LIN {X 266.912,Y -113.394,Z 120.558,A 156.982,B 90.000,C 0.000} C_DIS
LIN {X 267.031,Y -113.112,Z 120.601,A 157.043,B 90.000,C 0.000} C_DIS
LIN {X 267.056,Y -113.053,Z 120.652,A 157.056,B 90.000,C 0.000} C_DIS
LIN {X 267.089,Y -112.975,Z 120.703,A 157.072,B 90.000,C 0.000} C_DIS
LIN {X 267.248,Y -112.599,Z 120.745,A 157.153,B 90.000,C 0.000} C_DIS
LIN {X 267.281,Y -112.521,Z 120.796,A 157.170,B 90.000,C 0.000} C_DIS
LIN {X 267.306,Y -112.462,Z 120.847,A 157.182,B 90.000,C 0.000} C_DIS
LIN {X 267.424,Y -112.180,Z 120.890,A 157.243,B 90.000,C 0.000} C_DIS
LIN {X 267.449,Y -112.121,Z 120.941,A 157.255,B 90.000,C 0.000} C_DIS
LIN {X 267.482,Y -112.043,Z 120.992,A 157.272,B 90.000,C 0.000} C_DIS
LIN {X 267.639,Y -111.666,Z 121.034,A 157.353,B 90.000,C 0.000} C_DIS
LIN {X 267.705,Y -111.509,Z 121.137,A 157.386,B 90.000,C 0.000} C_DIS
LIN {X 267.861,Y -111.132,Z 121.179,A 157.467,B 90.000,C 0.000} C_DIS
LIN {X 267.894,Y -111.054,Z 121.230,A 157.484,B 90.000,C 0.000} C_DIS
LIN {X 267.918,Y -110.995,Z 121.281,A 157.496,B 90.000,C 0.000} C_DIS
LIN {X 268.035,Y -110.712,Z 121.324,A 157.557,B 90.000,C 0.000} C_DIS
LIN {X 268.060,Y -110.653,Z 121.375,A 157.570,B 90.000,C 0.000} C_DIS
LIN {X 268.092,Y -110.574,Z 121.426,A 157.586,B 90.000,C 0.000} C_DIS
LIN {X 268.247,Y -110.197,Z 121.468,A 157.667,B 90.000,C 0.000} C_DIS
LIN {X 268.312,Y -110.040,Z 121.570,A 157.701,B 90.000,C 0.000} C_DIS
LIN {X 268.466,Y -109.662,Z 121.613,A 157.781,B 90.000,C 0.000} C_DIS
LIN {X 268.499,Y -109.583,Z 121.664,A 157.798,B 90.000,C 0.000} C_DIS
LIN {X 268.523,Y -109.524,Z 121.715,A 157.811,B 90.000,C 0.000} C_DIS
LIN {X 268.638,Y -109.241,Z 121.757,A 157.871,B 90.000,C 0.000} C_DIS
LIN {X 268.662,Y -109.182,Z 121.808,A 157.884,B 90.000,C 0.000} C_DIS
LIN {X 268.694,Y -109.103,Z 121.859,A 157.900,B 90.000,C 0.000} C_DIS
LIN {X 268.847,Y -108.725,Z 121.902,A 157.981,B 90.000,C 0.000} C_DIS
LIN {X 268.879,Y -108.646,Z 121.953,A 157.998,B 90.000,C 0.000} C_DIS
LIN {X 268.899,Y -108.596,Z 122.004,A 158.009,B 90.000,C 0.000} C_DIS
LIN {X 269.023,Y -108.291,Z 122.077,A 158.074,B 90.000,C 0.000} C_DIS
LIN {X 269.087,Y -108.131,Z 122.214,A 158.108,B 90.000,C 0.000} C_DIS
LIN {X 269.132,Y -108.018,Z 122.410,A 158.132,B 90.000,C 0.000} C_DIS
LIN {X 269.157,Y -107.956,Z 122.817,A 158.145,B 90.000,C 0.000} C_DIS
LIN {X 269.176,Y -107.909,Z 122.892,A 158.155,B 90.000,C 0.000} C_DIS
LIN {X 269.195,Y -107.861,Z 123.037,A 158.165,B 90.000,C 0.000} C_DIS
LIN {X 269.211,Y -107.822,Z 123.759,A 158.173,B 90.000,C 0.000} C_DIS
LIN {X 269.249,Y -107.726,Z 124.048,A 158.194,B 90.000,C 0.000} C_DIS
LIN {X 269.264,Y -107.688,Z 124.771,A 158.202,B 90.000,C 0.000} C_DIS
LIN {X 269.303,Y -107.592,Z 125.060,A 158.222,B 90.000,C 0.000} C_DIS
LIN {X 269.318,Y -107.554,Z 125.783,A 158.230,B 90.000,C 0.000} C_DIS
LIN {X 269.356,Y -107.458,Z 126.072,A 158.251,B 90.000,C 0.000} C_DIS
LIN {X 269.372,Y -107.420,Z 126.794,A 158.259,B 90.000,C 0.000} C_DIS
LIN {X 269.391,Y -107.372,Z 126.939,A 158.269,B 90.000,C 0.000} C_DIS
LIN {X 269.410,Y -107.324,Z 127.003,A 158.279,B 90.000,C 0.000} C_DIS
LIN {X 269.431,Y -107.271,Z 127.336,A 158.291,B 90.000,C 0.000} C_DIS
LIN {X 269.498,Y -107.103,Z 127.372,A 158.326,B 90.000,C 0.000} C_DIS
LIN {X 269.554,Y -106.961,Z 127.351,A 158.356,B 90.000,C 0.000} C_DIS
LIN {X 269.601,Y -106.842,Z 127.249,A 158.382,B 90.000,C 0.000} C_DIS
LIN {X 269.714,Y -106.558,Z 127.207,A 158.442,B 90.000,C 0.000} C_DIS
LIN {X 269.760,Y -106.439,Z 127.105,A 158.467,B 90.000,C 0.000} C_DIS
LIN {X 269.873,Y -106.154,Z 127.062,A 158.528,B 90.000,C 0.000} C_DIS
LIN {X 269.896,Y -106.095,Z 127.011,A 158.540,B 90.000,C 0.000} C_DIS
LIN {X 269.911,Y -106.056,Z 126.960,A 158.549,B 90.000,C 0.000} C_DIS
LIN {X 269.986,Y -105.866,Z 126.918,A 158.589,B 90.000,C 0.000} C_DIS
LIN {X 270.002,Y -105.826,Z 126.867,A 158.598,B 90.000,C 0.000} C_DIS
LIN {X 270.025,Y -105.767,Z 126.816,A 158.610,B 90.000,C 0.000} C_DIS
LIN {X 270.136,Y -105.482,Z 126.773,A 158.671,B 90.000,C 0.000} C_DIS
LIN {X 270.183,Y -105.363,Z 126.671,A 158.696,B 90.000,C 0.000} C_DIS
LIN {X 270.294,Y -105.078,Z 126.629,A 158.756,B 90.000,C 0.000} C_DIS
LIN {X 270.340,Y -104.959,Z 126.527,A 158.781,B 90.000,C 0.000} C_DIS
LIN {X 270.451,Y -104.673,Z 126.484,A 158.842,B 90.000,C 0.000} C_DIS
LIN {X 270.474,Y -104.614,Z 126.433,A 158.854,B 90.000,C 0.000} C_DIS
LIN {X 270.486,Y -104.583,Z 126.382,A 158.861,B 90.000,C 0.000} C_DIS
LIN {X 270.514,Y -104.508,Z 126.361,A 158.877,B 90.000,C 0.000} C_DIS
LIN {X 270.595,Y -104.298,Z 126.250,A 158.921,B 90.000,C 0.000} C_DIS
LIN {X 270.620,Y -104.235,Z 126.135,A 158.935,B 90.000,C 0.000} C_DIS
LIN {X 270.542,Y -104.437,Z 125.878,A 158.892,B 90.000,C 0.000} C_DIS
LIN {X 270.518,Y -104.499,Z 125.673,A 158.879,B 90.000,C 0.000} C_DIS
LIN {X 270.481,Y -104.594,Z 125.596,A 158.859,B 90.000,C 0.000} C_DIS
LIN {X 270.466,Y -104.634,Z 125.392,A 158.850,B 90.000,C 0.000} C_DIS
LIN {X 270.429,Y -104.729,Z 125.307,A 158.830,B 90.000,C 0.000} C_DIS
LIN {X 270.414,Y -104.769,Z 125.102,A 158.822,B 90.000,C 0.000} C_DIS
LIN {X 270.377,Y -104.864,Z 125.018,A 158.802,B 90.000,C 0.000} C_DIS
LIN {X 270.361,Y -104.903,Z 124.813,A 158.793,B 90.000,C 0.000} C_DIS
LIN {X 270.324,Y -104.998,Z 124.728,A 158.773,B 90.000,C 0.000} C_DIS
LIN {X 270.309,Y -105.038,Z 124.524,A 158.765,B 90.000,C 0.000} C_DIS
LIN {X 270.291,Y -105.086,Z 124.482,A 158.755,B 90.000,C 0.000} C_DIS
LIN {X 270.272,Y -105.133,Z 124.418,A 158.744,B 90.000,C 0.000} C_DIS
LIN {X 270.257,Y -105.173,Z 124.112,A 158.736,B 90.000,C 0.000} C_DIS
LIN {X 270.220,Y -105.268,Z 123.985,A 158.716,B 90.000,C 0.000} C_DIS
LIN {X 270.204,Y -105.307,Z 123.678,A 158.708,B 90.000,C 0.000} C_DIS
LIN {X 270.167,Y -105.402,Z 123.551,A 158.687,B 90.000,C 0.000} C_DIS
LIN {X 270.152,Y -105.442,Z 123.245,A 158.679,B 90.000,C 0.000} C_DIS
LIN {X 270.133,Y -105.490,Z 123.181,A 158.669,B 90.000,C 0.000} C_DIS
LIN {X 270.115,Y -105.537,Z 123.075,A 158.659,B 90.000,C 0.000} C_DIS
LIN {X 270.099,Y -105.577,Z 122.565,A 158.650,B 90.000,C 0.000} C_DIS
LIN {X 270.081,Y -105.624,Z 122.458,A 158.640,B 90.000,C 0.000} C_DIS
LIN {X 270.061,Y -105.673,Z 122.242,A 158.630,B 90.000,C 0.000} C_DIS
LIN {X 270.047,Y -105.710,Z 121.085,A 158.622,B 90.000,C 0.000} C_DIS
LIN {X 270.028,Y -105.759,Z 120.869,A 158.612,B 90.000,C 0.000} C_DIS
LIN {X 270.009,Y -105.806,Z 120.805,A 158.602,B 90.000,C 0.000} C_DIS
LIN {X 270.002,Y -105.826,Z 120.652,A 158.598,B 90.000,C 0.000} C_DIS
LIN {X 270.009,Y -105.806,Z 120.499,A 158.602,B 90.000,C 0.000} C_DIS
LIN {X 270.028,Y -105.759,Z 120.435,A 158.612,B 90.000,C 0.000} C_DIS
LIN {X 270.047,Y -105.710,Z 120.236,A 158.622,B 90.000,C 0.000} C_DIS
LIN {X 270.062,Y -105.673,Z 119.189,A 158.630,B 90.000,C 0.000} C_DIS
LIN {X 270.081,Y -105.624,Z 118.990,A 158.640,B 90.000,C 0.000} C_DIS
LIN {X 270.099,Y -105.577,Z 118.884,A 158.650,B 90.000,C 0.000} C_DIS
LIN {X 270.115,Y -105.537,Z 118.373,A 158.659,B 90.000,C 0.000} C_DIS
LIN {X 270.152,Y -105.442,Z 118.182,A 158.679,B 90.000,C 0.000} C_DIS
LIN {X 270.167,Y -105.402,Z 117.774,A 158.687,B 90.000,C 0.000} C_DIS
LIN {X 270.186,Y -105.355,Z 117.689,A 158.697,B 90.000,C 0.000} C_DIS
LIN {X 270.204,Y -105.307,Z 117.625,A 158.708,B 90.000,C 0.000} C_DIS
LIN {X 270.220,Y -105.268,Z 117.319,A 158.716,B 90.000,C 0.000} C_DIS
LIN {X 270.238,Y -105.220,Z 117.255,A 158.726,B 90.000,C 0.000} C_DIS
LIN {X 270.257,Y -105.173,Z 117.213,A 158.736,B 90.000,C 0.000} C_DIS
LIN {X 270.272,Y -105.133,Z 117.009,A 158.744,B 90.000,C 0.000} C_DIS
LIN {X 270.291,Y -105.086,Z 116.966,A 158.755,B 90.000,C 0.000} C_DIS
LIN {X 270.309,Y -105.038,Z 116.903,A 158.765,B 90.000,C 0.000} C_DIS
LIN {X 270.324,Y -104.998,Z 116.597,A 158.773,B 90.000,C 0.000} C_DIS
LIN {X 270.343,Y -104.951,Z 116.533,A 158.783,B 90.000,C 0.000} C_DIS
LIN {X 270.361,Y -104.903,Z 116.490,A 158.793,B 90.000,C 0.000} C_DIS
LIN {X 270.377,Y -104.864,Z 116.286,A 158.802,B 90.000,C 0.000} C_DIS
LIN {X 270.414,Y -104.769,Z 116.201,A 158.822,B 90.000,C 0.000} C_DIS
LIN {X 270.429,Y -104.729,Z 115.997,A 158.830,B 90.000,C 0.000} C_DIS
LIN {X 270.466,Y -104.634,Z 115.917,A 158.850,B 90.000,C 0.000} C_DIS
LIN {X 270.474,Y -104.614,Z 115.826,A 158.854,B 90.000,C 0.000} C_DIS
LIN {X 270.489,Y -104.574,Z 115.705,A 158.863,B 90.000,C 0.000} C_DIS
LIN {X 270.562,Y -104.384,Z 115.487,A 158.903,B 90.000,C 0.000} C_DIS
LIN {X 270.593,Y -104.305,Z 115.266,A 158.920,B 90.000,C 0.000} C_DIS
LIN {X 270.666,Y -104.114,Z 115.053,A 158.960,B 90.000,C 0.000} C_DIS
LIN {X 270.697,Y -104.035,Z 114.833,A 158.977,B 90.000,C 0.000} C_DIS
LIN {X 270.733,Y -103.940,Z 114.726,A 158.997,B 90.000,C 0.000} C_DIS
LIN {X 271.344,Y -102.334,Z 112.910,A 159.337,B 90.000,C 0.000} C_DIS
LIN {X 271.563,Y -101.752,Z 112.405,A 159.460,B 90.000,C 0.000} C_DIS
LIN {X 271.644,Y -101.535,Z 112.299,A 159.505,B 90.000,C 0.000} C_DIS
LIN {X 271.719,Y -101.335,Z 112.095,A 159.548,B 90.000,C 0.000} C_DIS
LIN {X 271.761,Y -101.221,Z 112.052,A 159.572,B 90.000,C 0.000} C_DIS
LIN {X 271.793,Y -101.136,Z 112.031,A 159.589,B 90.000,C 0.000} C_DIS
LIN {X 271.820,Y -101.065,Z 111.929,A 159.604,B 90.000,C 0.000} C_DIS
LIN {X 271.851,Y -100.980,Z 111.908,A 159.622,B 90.000,C 0.000} C_DIS
LIN {X 271.893,Y -100.866,Z 111.865,A 159.646,B 90.000,C 0.000} C_DIS
LIN {X 271.971,Y -100.657,Z 111.661,A 159.690,B 90.000,C 0.000} C_DIS
LIN {X 272.013,Y -100.544,Z 111.619,A 159.714,B 90.000,C 0.000} C_DIS
LIN {X 272.044,Y -100.458,Z 111.598,A 159.732,B 90.000,C 0.000} C_DIS
LIN {X 272.057,Y -100.423,Z 111.547,A 159.740,B 90.000,C 0.000} C_DIS
LIN {X 272.079,Y -100.363,Z 111.496,A 159.752,B 90.000,C 0.000} C_DIS
LIN {X 272.185,Y -100.076,Z 111.453,A 159.813,B 90.000,C 0.000} C_DIS
LIN {X 272.207,Y -100.016,Z 111.402,A 159.825,B 90.000,C 0.000} C_DIS
LIN {X 272.222,Y -99.976,Z 111.351,A 159.834,B 90.000,C 0.000} C_DIS
LIN {X 272.292,Y -99.785,Z 111.309,A 159.874,B 90.000,C 0.000} C_DIS
LIN {X 272.307,Y -99.745,Z 111.258,A 159.882,B 90.000,C 0.000} C_DIS
LIN {X 272.329,Y -99.685,Z 111.207,A 159.895,B 90.000,C 0.000} C_DIS
LIN {X 272.434,Y -99.397,Z 111.164,A 159.956,B 90.000,C 0.000} C_DIS
LIN {X 272.477,Y -99.278,Z 111.062,A 159.981,B 90.000,C 0.000} C_DIS
LIN {X 272.582,Y -98.990,Z 111.020,A 160.041,B 90.000,C 0.000} C_DIS
LIN {X 272.604,Y -98.930,Z 110.969,A 160.054,B 90.000,C 0.000} C_DIS
LIN {X 272.633,Y -98.850,Z 110.917,A 160.071,B 90.000,C 0.000} C_DIS
LIN {X 272.772,Y -98.466,Z 110.875,A 160.151,B 90.000,C 0.000} C_DIS
LIN {X 272.801,Y -98.386,Z 110.824,A 160.168,B 90.000,C 0.000} C_DIS
LIN {X 272.843,Y -98.267,Z 110.773,A 160.193,B 90.000,C 0.000} C_DIS
LIN {X 273.051,Y -97.689,Z 110.731,A 160.314,B 90.000,C 0.000} C_DIS
LIN {X 273.094,Y -97.570,Z 110.679,A 160.339,B 90.000,C 0.000} C_DIS
LIN {X 273.215,Y -97.230,Z 110.626,A 160.411,B 90.000,C 0.000} C_DIS
LIN {X 273.887,Y -95.321,Z 110.626,A 160.810,B 90.000,C 0.000} C_DIS
LIN {X 274.005,Y -94.980,Z 110.679,A 160.882,B 90.000,C 0.000} C_DIS
LIN {X 274.047,Y -94.860,Z 110.731,A 160.907,B 90.000,C 0.000} C_DIS
LIN {X 274.247,Y -94.280,Z 110.773,A 161.028,B 90.000,C 0.000} C_DIS
LIN {X 274.288,Y -94.160,Z 110.824,A 161.053,B 90.000,C 0.000} C_DIS
LIN {X 274.316,Y -94.080,Z 110.875,A 161.070,B 90.000,C 0.000} C_DIS
LIN {X 274.448,Y -93.693,Z 110.917,A 161.151,B 90.000,C 0.000} C_DIS
LIN {X 274.475,Y -93.613,Z 110.969,A 161.167,B 90.000,C 0.000} C_DIS
LIN {X 274.496,Y -93.553,Z 111.020,A 161.180,B 90.000,C 0.000} C_DIS
LIN {X 274.594,Y -93.263,Z 111.062,A 161.241,B 90.000,C 0.000} C_DIS
LIN {X 274.635,Y -93.142,Z 111.164,A 161.266,B 90.000,C 0.000} C_DIS
LIN {X 274.733,Y -92.852,Z 111.207,A 161.326,B 90.000,C 0.000} C_DIS
LIN {X 274.754,Y -92.792,Z 111.258,A 161.339,B 90.000,C 0.000} C_DIS
LIN {X 274.767,Y -92.752,Z 111.309,A 161.347,B 90.000,C 0.000} C_DIS
LIN {X 274.833,Y -92.558,Z 111.351,A 161.387,B 90.000,C 0.000} C_DIS
LIN {X 274.846,Y -92.518,Z 111.402,A 161.396,B 90.000,C 0.000} C_DIS
LIN {X 274.866,Y -92.458,Z 111.453,A 161.408,B 90.000,C 0.000} C_DIS
LIN {X 274.964,Y -92.167,Z 111.496,A 161.469,B 90.000,C 0.000} C_DIS
LIN {X 274.984,Y -92.107,Z 111.547,A 161.482,B 90.000,C 0.000} C_DIS
LIN {X 274.996,Y -92.071,Z 111.598,A 161.489,B 90.000,C 0.000} C_DIS
LIN {X 275.025,Y -91.985,Z 111.619,A 161.507,B 90.000,C 0.000} C_DIS
LIN {X 275.063,Y -91.870,Z 111.661,A 161.531,B 90.000,C 0.000} C_DIS
LIN {X 275.134,Y -91.659,Z 111.865,A 161.575,B 90.000,C 0.000} C_DIS
LIN {X 275.172,Y -91.544,Z 111.908,A 161.599,B 90.000,C 0.000} C_DIS
LIN {X 275.201,Y -91.457,Z 111.929,A 161.617,B 90.000,C 0.000} C_DIS
LIN {X 275.225,Y -91.386,Z 112.031,A 161.632,B 90.000,C 0.000} C_DIS
LIN {X 275.253,Y -91.299,Z 112.052,A 161.650,B 90.000,C 0.000} C_DIS
LIN {X 275.292,Y -91.184,Z 112.095,A 161.674,B 90.000,C 0.000} C_DIS
LIN {X 275.360,Y -90.977,Z 112.299,A 161.717,B 90.000,C 0.000} C_DIS
LIN {X 275.429,Y -90.768,Z 112.384,A 161.760,B 90.000,C 0.000} C_DIS
LIN {X 275.462,Y -90.667,Z 112.486,A 161.781,B 90.000,C 0.000} C_DIS
LIN {X 276.031,Y -88.920,Z 114.182,A 162.144,B 90.000,C 0.000} C_DIS
LIN {X 276.087,Y -88.747,Z 114.365,A 162.180,B 90.000,C 0.000} C_DIS
LIN {X 276.676,Y -86.892,Z 114.346,A 162.565,B 90.000,C 0.000} C_DIS
LIN {X 276.857,Y -86.314,Z 114.239,A 162.684,B 90.000,C 0.000} C_DIS
LIN {X 277.358,Y -84.691,Z 114.201,A 163.020,B 90.000,C 0.000} C_DIS
LIN {X 277.537,Y -84.104,Z 114.095,A 163.141,B 90.000,C 0.000} C_DIS
LIN {X 278.024,Y -82.477,Z 114.057,A 163.477,B 90.000,C 0.000} C_DIS
LIN {X 278.198,Y -81.888,Z 113.950,A 163.598,B 90.000,C 0.000} C_DIS
LIN {X 278.673,Y -80.258,Z 113.912,A 163.934,B 90.000,C 0.000} C_DIS
LIN {X 278.843,Y -79.667,Z 113.806,A 164.055,B 90.000,C 0.000} C_DIS
LIN {X 279.304,Y -78.033,Z 113.767,A 164.391,B 90.000,C 0.000} C_DIS
LIN {X 279.469,Y -77.441,Z 113.661,A 164.512,B 90.000,C 0.000} C_DIS
LIN {X 279.918,Y -75.803,Z 113.661,A 164.847,B 90.000,C 0.000} C_DIS
LIN {X 279.998,Y -75.507,Z 113.714,A 164.908,B 90.000,C 0.000} C_DIS
LIN {X 280.006,Y -75.475,Z 113.765,A 164.915,B 90.000,C 0.000} C_DIS
LIN {X 280.027,Y -75.400,Z 113.787,A 164.930,B 90.000,C 0.000} C_DIS
LIN {X 280.065,Y -75.256,Z 113.860,A 164.959,B 90.000,C 0.000} C_DIS
LIN {X 280.118,Y -75.059,Z 114.032,A 165.000,B 90.000,C 0.000} C_DIS
LIN {X 280.165,Y -74.884,Z 114.225,A 165.035,B 90.000,C 0.000} C_DIS
LIN {X 280.199,Y -74.756,Z 114.483,A 165.062,B 90.000,C 0.000} C_DIS
LIN {X 280.233,Y -74.630,Z 114.626,A 165.088,B 90.000,C 0.000} C_DIS
LIN {X 280.273,Y -74.480,Z 114.747,A 165.118,B 90.000,C 0.000} C_DIS
LIN {X 280.305,Y -74.358,Z 114.798,A 165.143,B 90.000,C 0.000} C_DIS
LIN {X 280.325,Y -74.282,Z 114.777,A 165.159,B 90.000,C 0.000} C_DIS
LIN {X 280.334,Y -74.250,Z 114.726,A 165.165,B 90.000,C 0.000} C_DIS
LIN {X 280.344,Y -74.209,Z 114.675,A 165.173,B 90.000,C 0.000} C_DIS
LIN {X 280.397,Y -74.012,Z 114.633,A 165.214,B 90.000,C 0.000} C_DIS
LIN {X 280.407,Y -73.971,Z 114.582,A 165.222,B 90.000,C 0.000} C_DIS
LIN {X 280.424,Y -73.909,Z 114.531,A 165.235,B 90.000,C 0.000} C_DIS
LIN {X 280.502,Y -73.613,Z 114.488,A 165.295,B 90.000,C 0.000} C_DIS
LIN {X 280.534,Y -73.490,Z 114.386,A 165.320,B 90.000,C 0.000} C_DIS
LIN {X 280.611,Y -73.193,Z 114.344,A 165.381,B 90.000,C 0.000} C_DIS
LIN {X 280.643,Y -73.070,Z 114.241,A 165.406,B 90.000,C 0.000} C_DIS
LIN {X 280.720,Y -72.774,Z 114.199,A 165.467,B 90.000,C 0.000} C_DIS
LIN {X 280.736,Y -72.712,Z 114.148,A 165.479,B 90.000,C 0.000} C_DIS
LIN {X 280.747,Y -72.671,Z 114.097,A 165.488,B 90.000,C 0.000} C_DIS
LIN {X 280.798,Y -72.473,Z 114.054,A 165.528,B 90.000,C 0.000} C_DIS
LIN {X 280.809,Y -72.432,Z 114.003,A 165.536,B 90.000,C 0.000} C_DIS
LIN {X 280.825,Y -72.371,Z 113.952,A 165.549,B 90.000,C 0.000} C_DIS
LIN {X 280.901,Y -72.074,Z 113.910,A 165.609,B 90.000,C 0.000} C_DIS
LIN {X 280.933,Y -71.951,Z 113.808,A 165.635,B 90.000,C 0.000} C_DIS
LIN {X 281.008,Y -71.654,Z 113.765,A 165.695,B 90.000,C 0.000} C_DIS
LIN {X 281.040,Y -71.531,Z 113.663,A 165.720,B 90.000,C 0.000} C_DIS
LIN {X 281.115,Y -71.234,Z 113.621,A 165.781,B 90.000,C 0.000} C_DIS
LIN {X 281.131,Y -71.172,Z 113.570,A 165.793,B 90.000,C 0.000} C_DIS
LIN {X 281.141,Y -71.131,Z 113.519,A 165.802,B 90.000,C 0.000} C_DIS
LIN {X 281.191,Y -70.933,Z 113.476,A 165.842,B 90.000,C 0.000} C_DIS
LIN {X 281.202,Y -70.892,Z 113.425,A 165.850,B 90.000,C 0.000} C_DIS
LIN {X 281.217,Y -70.830,Z 113.374,A 165.863,B 90.000,C 0.000} C_DIS
LIN {X 281.292,Y -70.533,Z 113.332,A 165.923,B 90.000,C 0.000} C_DIS
LIN {X 281.323,Y -70.410,Z 113.230,A 165.949,B 90.000,C 0.000} C_DIS
LIN {X 281.397,Y -70.112,Z 113.187,A 166.009,B 90.000,C 0.000} C_DIS
LIN {X 281.428,Y -69.989,Z 113.085,A 166.034,B 90.000,C 0.000} C_DIS
LIN {X 281.501,Y -69.692,Z 113.043,A 166.095,B 90.000,C 0.000} C_DIS
LIN {X 281.517,Y -69.630,Z 112.992,A 166.107,B 90.000,C 0.000} C_DIS
LIN {X 281.527,Y -69.589,Z 112.941,A 166.116,B 90.000,C 0.000} C_DIS
LIN {X 281.576,Y -69.390,Z 112.898,A 166.156,B 90.000,C 0.000} C_DIS
LIN {X 281.586,Y -69.349,Z 112.847,A 166.164,B 90.000,C 0.000} C_DIS
LIN {X 281.601,Y -69.287,Z 112.796,A 166.177,B 90.000,C 0.000} C_DIS
LIN {X 281.674,Y -68.990,Z 112.754,A 166.238,B 90.000,C 0.000} C_DIS
LIN {X 281.705,Y -68.866,Z 112.652,A 166.263,B 90.000,C 0.000} C_DIS
LIN {X 281.777,Y -68.569,Z 112.609,A 166.323,B 90.000,C 0.000} C_DIS
LIN {X 281.792,Y -68.507,Z 112.558,A 166.336,B 90.000,C 0.000} C_DIS
LIN {X 281.802,Y -68.466,Z 112.507,A 166.344,B 90.000,C 0.000} C_DIS
LIN {X 281.850,Y -68.267,Z 112.465,A 166.385,B 90.000,C 0.000} C_DIS
LIN {X 281.860,Y -68.226,Z 112.414,A 166.393,B 90.000,C 0.000} C_DIS
LIN {X 281.875,Y -68.164,Z 112.363,A 166.406,B 90.000,C 0.000} C_DIS
LIN {X 281.947,Y -67.866,Z 112.320,A 166.466,B 90.000,C 0.000} C_DIS
LIN {X 281.977,Y -67.743,Z 112.218,A 166.491,B 90.000,C 0.000} C_DIS
LIN {X 282.048,Y -67.445,Z 112.176,A 166.552,B 90.000,C 0.000} C_DIS
LIN {X 282.078,Y -67.321,Z 112.074,A 166.577,B 90.000,C 0.000} C_DIS
LIN {X 282.149,Y -67.023,Z 112.031,A 166.637,B 90.000,C 0.000} C_DIS
LIN {X 282.163,Y -66.961,Z 111.980,A 166.650,B 90.000,C 0.000} C_DIS
LIN {X 282.173,Y -66.920,Z 111.929,A 166.658,B 90.000,C 0.000} C_DIS
LIN {X 282.220,Y -66.721,Z 111.887,A 166.699,B 90.000,C 0.000} C_DIS
LIN {X 282.230,Y -66.680,Z 111.836,A 166.707,B 90.000,C 0.000} C_DIS
LIN {X 282.245,Y -66.618,Z 111.784,A 166.720,B 90.000,C 0.000} C_DIS
LIN {X 282.315,Y -66.320,Z 111.742,A 166.780,B 90.000,C 0.000} C_DIS
LIN {X 282.344,Y -66.196,Z 111.640,A 166.805,B 90.000,C 0.000} C_DIS
LIN {X 282.414,Y -65.898,Z 111.597,A 166.866,B 90.000,C 0.000} C_DIS
LIN {X 282.443,Y -65.774,Z 111.495,A 166.891,B 90.000,C 0.000} C_DIS
LIN {X 282.512,Y -65.475,Z 111.453,A 166.951,B 90.000,C 0.000} C_DIS
LIN {X 282.526,Y -65.413,Z 111.402,A 166.964,B 90.000,C 0.000} C_DIS
LIN {X 282.536,Y -65.372,Z 111.351,A 166.972,B 90.000,C 0.000} C_DIS
LIN {X 282.582,Y -65.173,Z 111.308,A 167.013,B 90.000,C 0.000} C_DIS
LIN {X 282.591,Y -65.132,Z 111.257,A 167.021,B 90.000,C 0.000} C_DIS
LIN {X 282.606,Y -65.070,Z 111.206,A 167.034,B 90.000,C 0.000} C_DIS
LIN {X 282.674,Y -64.771,Z 111.164,A 167.094,B 90.000,C 0.000} C_DIS
LIN {X 282.703,Y -64.647,Z 111.062,A 167.119,B 90.000,C 0.000} C_DIS
LIN {X 282.771,Y -64.348,Z 111.019,A 167.180,B 90.000,C 0.000} C_DIS
LIN {X 282.785,Y -64.286,Z 110.968,A 167.192,B 90.000,C 0.000} C_DIS
LIN {X 282.794,Y -64.245,Z 110.917,A 167.201,B 90.000,C 0.000} C_DIS
LIN {X 282.839,Y -64.046,Z 110.875,A 167.241,B 90.000,C 0.000} C_DIS
LIN {X 282.849,Y -64.004,Z 110.824,A 167.250,B 90.000,C 0.000} C_DIS
LIN {X 282.863,Y -63.942,Z 110.773,A 167.262,B 90.000,C 0.000} C_DIS
LIN {X 282.930,Y -63.644,Z 110.730,A 167.323,B 90.000,C 0.000} C_DIS
LIN {X 282.958,Y -63.519,Z 110.628,A 167.348,B 90.000,C 0.000} C_DIS
LIN {X 283.025,Y -63.220,Z 110.586,A 167.408,B 90.000,C 0.000} C_DIS
LIN {X 283.053,Y -63.096,Z 110.484,A 167.433,B 90.000,C 0.000} C_DIS
LIN {X 283.119,Y -62.797,Z 110.441,A 167.494,B 90.000,C 0.000} C_DIS
LIN {X 283.133,Y -62.735,Z 110.390,A 167.507,B 90.000,C 0.000} C_DIS
LIN {X 283.142,Y -62.694,Z 110.339,A 167.515,B 90.000,C 0.000} C_DIS
LIN {X 283.186,Y -62.494,Z 110.297,A 167.555,B 90.000,C 0.000} C_DIS
LIN {X 283.195,Y -62.453,Z 110.246,A 167.564,B 90.000,C 0.000} C_DIS
LIN {X 283.209,Y -62.391,Z 110.195,A 167.576,B 90.000,C 0.000} C_DIS
LIN {X 283.275,Y -62.092,Z 110.152,A 167.637,B 90.000,C 0.000} C_DIS
LIN {X 283.302,Y -61.967,Z 110.050,A 167.662,B 90.000,C 0.000} C_DIS
LIN {X 283.367,Y -61.668,Z 110.008,A 167.722,B 90.000,C 0.000} C_DIS
LIN {X 283.394,Y -61.543,Z 109.906,A 167.748,B 90.000,C 0.000} C_DIS
LIN {X 283.459,Y -61.244,Z 109.863,A 167.808,B 90.000,C 0.000} C_DIS
LIN {X 283.473,Y -61.182,Z 109.812,A 167.821,B 90.000,C 0.000} C_DIS
LIN {X 283.482,Y -61.140,Z 109.761,A 167.829,B 90.000,C 0.000} C_DIS
LIN {X 283.525,Y -60.941,Z 109.719,A 167.869,B 90.000,C 0.000} C_DIS
LIN {X 283.534,Y -60.899,Z 109.668,A 167.878,B 90.000,C 0.000} C_DIS
LIN {X 283.547,Y -60.837,Z 109.617,A 167.890,B 90.000,C 0.000} C_DIS
LIN {X 283.611,Y -60.538,Z 109.574,A 167.951,B 90.000,C 0.000} C_DIS
LIN {X 283.638,Y -60.413,Z 109.472,A 167.976,B 90.000,C 0.000} C_DIS
LIN {X 283.701,Y -60.114,Z 109.430,A 168.037,B 90.000,C 0.000} C_DIS
LIN {X 283.714,Y -60.051,Z 109.379,A 168.049,B 90.000,C 0.000} C_DIS
LIN {X 283.723,Y -60.010,Z 109.328,A 168.057,B 90.000,C 0.000} C_DIS
LIN {X 283.765,Y -59.810,Z 109.285,A 168.098,B 90.000,C 0.000} C_DIS
LIN {X 283.774,Y -59.768,Z 109.234,A 168.106,B 90.000,C 0.000} C_DIS
LIN {X 283.787,Y -59.706,Z 109.183,A 168.119,B 90.000,C 0.000} C_DIS
LIN {X 283.850,Y -59.406,Z 109.141,A 168.179,B 90.000,C 0.000} C_DIS
LIN {X 283.876,Y -59.282,Z 109.038,A 168.204,B 90.000,C 0.000} C_DIS
LIN {X 283.939,Y -58.982,Z 108.996,A 168.265,B 90.000,C 0.000} C_DIS
LIN {X 283.964,Y -58.857,Z 108.894,A 168.290,B 90.000,C 0.000} C_DIS
LIN {X 284.026,Y -58.557,Z 108.851,A 168.351,B 90.000,C 0.000} C_DIS
LIN {X 284.039,Y -58.495,Z 108.800,A 168.363,B 90.000,C 0.000} C_DIS
LIN {X 284.048,Y -58.453,Z 108.749,A 168.372,B 90.000,C 0.000} C_DIS
LIN {X 284.089,Y -58.253,Z 108.707,A 168.412,B 90.000,C 0.000} C_DIS
LIN {X 284.097,Y -58.212,Z 108.656,A 168.420,B 90.000,C 0.000} C_DIS
LIN {X 284.110,Y -58.149,Z 108.605,A 168.433,B 90.000,C 0.000} C_DIS
LIN {X 284.172,Y -57.849,Z 108.562,A 168.493,B 90.000,C 0.000} C_DIS
LIN {X 284.197,Y -57.725,Z 108.460,A 168.519,B 90.000,C 0.000} C_DIS
LIN {X 284.258,Y -57.425,Z 108.418,A 168.579,B 90.000,C 0.000} C_DIS
LIN {X 284.283,Y -57.300,Z 108.316,A 168.604,B 90.000,C 0.000} C_DIS
LIN {X 284.343,Y -56.999,Z 108.273,A 168.665,B 90.000,C 0.000} C_DIS
LIN {X 284.356,Y -56.937,Z 108.222,A 168.677,B 90.000,C 0.000} C_DIS
LIN {X 284.364,Y -56.895,Z 108.171,A 168.686,B 90.000,C 0.000} C_DIS
LIN {X 284.404,Y -56.695,Z 108.129,A 168.726,B 90.000,C 0.000} C_DIS
LIN {X 284.412,Y -56.654,Z 108.078,A 168.734,B 90.000,C 0.000} C_DIS
LIN {X 284.425,Y -56.591,Z 108.027,A 168.747,B 90.000,C 0.000} C_DIS
LIN {X 284.484,Y -56.291,Z 107.984,A 168.808,B 90.000,C 0.000} C_DIS
LIN {X 284.509,Y -56.166,Z 107.882,A 168.833,B 90.000,C 0.000} C_DIS
LIN {X 284.568,Y -55.865,Z 107.840,A 168.893,B 90.000,C 0.000} C_DIS
LIN {X 284.580,Y -55.803,Z 107.789,A 168.906,B 90.000,C 0.000} C_DIS
LIN {X 284.589,Y -55.761,Z 107.738,A 168.914,B 90.000,C 0.000} C_DIS
LIN {X 284.628,Y -55.561,Z 107.695,A 168.954,B 90.000,C 0.000} C_DIS
LIN {X 284.636,Y -55.519,Z 107.644,A 168.963,B 90.000,C 0.000} C_DIS
LIN {X 284.648,Y -55.457,Z 107.593,A 168.975,B 90.000,C 0.000} C_DIS
LIN {X 284.707,Y -55.156,Z 107.551,A 169.036,B 90.000,C 0.000} C_DIS
LIN {X 284.731,Y -55.031,Z 107.449,A 169.061,B 90.000,C 0.000} C_DIS
LIN {X 284.789,Y -54.730,Z 107.406,A 169.122,B 90.000,C 0.000} C_DIS
LIN {X 284.813,Y -54.605,Z 107.304,A 169.147,B 90.000,C 0.000} C_DIS
LIN {X 284.870,Y -54.304,Z 107.262,A 169.207,B 90.000,C 0.000} C_DIS
LIN {X 284.882,Y -54.242,Z 107.211,A 169.220,B 90.000,C 0.000} C_DIS
LIN {X 284.890,Y -54.200,Z 107.160,A 169.228,B 90.000,C 0.000} C_DIS
LIN {X 284.928,Y -54.000,Z 107.117,A 169.269,B 90.000,C 0.000} C_DIS
LIN {X 284.936,Y -53.958,Z 107.066,A 169.277,B 90.000,C 0.000} C_DIS
LIN {X 284.948,Y -53.895,Z 107.015,A 169.290,B 90.000,C 0.000} C_DIS
LIN {X 285.005,Y -53.594,Z 106.973,A 169.350,B 90.000,C 0.000} C_DIS
LIN {X 285.028,Y -53.469,Z 106.871,A 169.375,B 90.000,C 0.000} C_DIS
LIN {X 285.084,Y -53.168,Z 106.828,A 169.436,B 90.000,C 0.000} C_DIS
LIN {X 285.108,Y -53.043,Z 106.726,A 169.461,B 90.000,C 0.000} C_DIS
LIN {X 285.164,Y -52.742,Z 106.684,A 169.521,B 90.000,C 0.000} C_DIS
LIN {X 285.175,Y -52.679,Z 106.633,A 169.534,B 90.000,C 0.000} C_DIS
LIN {X 285.183,Y -52.638,Z 106.581,A 169.542,B 90.000,C 0.000} C_DIS
LIN {X 285.220,Y -52.437,Z 106.539,A 169.583,B 90.000,C 0.000} C_DIS
LIN {X 285.228,Y -52.395,Z 106.488,A 169.591,B 90.000,C 0.000} C_DIS
LIN {X 285.239,Y -52.332,Z 106.437,A 169.604,B 90.000,C 0.000} C_DIS
LIN {X 285.294,Y -52.031,Z 106.394,A 169.664,B 90.000,C 0.000} C_DIS
LIN {X 285.317,Y -51.906,Z 106.292,A 169.689,B 90.000,C 0.000} C_DIS
LIN {X 285.372,Y -51.605,Z 106.250,A 169.750,B 90.000,C 0.000} C_DIS
LIN {X 285.394,Y -51.479,Z 106.148,A 169.775,B 90.000,C 0.000} C_DIS
LIN {X 285.448,Y -51.178,Z 106.105,A 169.835,B 90.000,C 0.000} C_DIS
LIN {X 285.460,Y -51.115,Z 106.054,A 169.848,B 90.000,C 0.000} C_DIS
LIN {X 285.467,Y -51.073,Z 106.003,A 169.856,B 90.000,C 0.000} C_DIS
LIN {X 285.503,Y -50.872,Z 105.961,A 169.897,B 90.000,C 0.000} C_DIS
LIN {X 285.511,Y -50.831,Z 105.910,A 169.905,B 90.000,C 0.000} C_DIS
LIN {X 285.522,Y -50.768,Z 105.859,A 169.918,B 90.000,C 0.000} C_DIS
LIN {X 285.575,Y -50.466,Z 105.816,A 169.978,B 90.000,C 0.000} C_DIS
LIN {X 285.597,Y -50.341,Z 105.714,A 170.003,B 90.000,C 0.000} C_DIS
LIN {X 285.650,Y -50.039,Z 105.672,A 170.064,B 90.000,C 0.000} C_DIS
LIN {X 285.672,Y -49.914,Z 105.570,A 170.089,B 90.000,C 0.000} C_DIS
LIN {X 285.725,Y -49.612,Z 105.527,A 170.150,B 90.000,C 0.000} C_DIS
LIN {X 285.736,Y -49.550,Z 105.476,A 170.162,B 90.000,C 0.000} C_DIS
LIN {X 285.743,Y -49.508,Z 105.425,A 170.171,B 90.000,C 0.000} C_DIS
LIN {X 285.778,Y -49.307,Z 105.383,A 170.211,B 90.000,C 0.000} C_DIS
LIN {X 285.785,Y -49.265,Z 105.332,A 170.219,B 90.000,C 0.000} C_DIS
LIN {X 285.796,Y -49.202,Z 105.281,A 170.232,B 90.000,C 0.000} C_DIS
LIN {X 285.847,Y -48.900,Z 105.238,A 170.292,B 90.000,C 0.000} C_DIS
LIN {X 285.869,Y -48.775,Z 105.136,A 170.318,B 90.000,C 0.000} C_DIS
LIN {X 285.920,Y -48.473,Z 105.094,A 170.378,B 90.000,C 0.000} C_DIS
LIN {X 285.931,Y -48.410,Z 105.043,A 170.391,B 90.000,C 0.000} C_DIS
LIN {X 285.938,Y -48.368,Z 104.992,A 170.399,B 90.000,C 0.000} C_DIS
LIN {X 285.972,Y -48.167,Z 104.949,A 170.439,B 90.000,C 0.000} C_DIS
LIN {X 285.979,Y -48.125,Z 104.898,A 170.448,B 90.000,C 0.000} C_DIS
LIN {X 285.990,Y -48.062,Z 104.847,A 170.460,B 90.000,C 0.000} C_DIS
LIN {X 286.040,Y -47.760,Z 104.805,A 170.521,B 90.000,C 0.000} C_DIS
LIN {X 286.061,Y -47.634,Z 104.703,A 170.546,B 90.000,C 0.000} C_DIS
LIN {X 286.111,Y -47.332,Z 104.660,A 170.606,B 90.000,C 0.000} C_DIS
LIN {X 286.132,Y -47.207,Z 104.558,A 170.632,B 90.000,C 0.000} C_DIS
LIN {X 286.182,Y -46.905,Z 104.516,A 170.692,B 90.000,C 0.000} C_DIS
LIN {X 286.192,Y -46.842,Z 104.465,A 170.705,B 90.000,C 0.000} C_DIS
LIN {X 286.199,Y -46.800,Z 104.414,A 170.713,B 90.000,C 0.000} C_DIS
LIN {X 286.232,Y -46.598,Z 104.371,A 170.753,B 90.000,C 0.000} C_DIS
LIN {X 286.239,Y -46.556,Z 104.320,A 170.762,B 90.000,C 0.000} C_DIS
LIN {X 286.249,Y -46.494,Z 104.269,A 170.774,B 90.000,C 0.000} C_DIS
LIN {X 286.298,Y -46.191,Z 104.227,A 170.835,B 90.000,C 0.000} C_DIS
LIN {X 286.318,Y -46.065,Z 104.124,A 170.860,B 90.000,C 0.000} C_DIS
LIN {X 286.366,Y -45.763,Z 104.082,A 170.921,B 90.000,C 0.000} C_DIS
LIN {X 286.387,Y -45.637,Z 103.980,A 170.946,B 90.000,C 0.000} C_DIS
LIN {X 286.435,Y -45.335,Z 103.938,A 171.006,B 90.000,C 0.000} C_DIS
LIN {X 286.444,Y -45.272,Z 103.886,A 171.019,B 90.000,C 0.000} C_DIS
LIN {X 286.451,Y -45.230,Z 103.835,A 171.027,B 90.000,C 0.000} C_DIS
LIN {X 286.483,Y -45.028,Z 103.793,A 171.068,B 90.000,C 0.000} C_DIS
LIN {X 286.489,Y -44.987,Z 103.742,A 171.076,B 90.000,C 0.000} C_DIS
LIN {X 286.499,Y -44.924,Z 103.691,A 171.088,B 90.000,C 0.000} C_DIS
LIN {X 286.547,Y -44.621,Z 103.648,A 171.149,B 90.000,C 0.000} C_DIS
LIN {X 286.566,Y -44.495,Z 103.546,A 171.174,B 90.000,C 0.000} C_DIS
LIN {X 286.613,Y -44.193,Z 103.504,A 171.235,B 90.000,C 0.000} C_DIS
LIN {X 286.623,Y -44.130,Z 103.453,A 171.247,B 90.000,C 0.000} C_DIS
LIN {X 286.629,Y -44.088,Z 103.402,A 171.256,B 90.000,C 0.000} C_DIS
LIN {X 286.660,Y -43.886,Z 103.359,A 171.296,B 90.000,C 0.000} C_DIS
LIN {X 286.667,Y -43.844,Z 103.308,A 171.304,B 90.000,C 0.000} C_DIS
LIN {X 286.676,Y -43.781,Z 103.257,A 171.317,B 90.000,C 0.000} C_DIS
LIN {X 286.722,Y -43.478,Z 103.215,A 171.377,B 90.000,C 0.000} C_DIS
LIN {X 286.741,Y -43.352,Z 103.113,A 171.403,B 90.000,C 0.000} C_DIS
LIN {X 286.787,Y -43.049,Z 103.070,A 171.463,B 90.000,C 0.000} C_DIS
LIN {X 286.806,Y -42.924,Z 102.968,A 171.488,B 90.000,C 0.000} C_DIS
LIN {X 286.851,Y -42.621,Z 102.926,A 171.549,B 90.000,C 0.000} C_DIS
LIN {X 286.860,Y -42.558,Z 102.875,A 171.561,B 90.000,C 0.000} C_DIS
LIN {X 286.867,Y -42.516,Z 102.824,A 171.570,B 90.000,C 0.000} C_DIS
LIN {X 286.896,Y -42.314,Z 102.781,A 171.610,B 90.000,C 0.000} C_DIS
LIN {X 286.903,Y -42.272,Z 102.730,A 171.618,B 90.000,C 0.000} C_DIS
LIN {X 286.912,Y -42.209,Z 102.679,A 171.631,B 90.000,C 0.000} C_DIS
LIN {X 286.956,Y -41.906,Z 102.637,A 171.692,B 90.000,C 0.000} C_DIS
LIN {X 286.975,Y -41.780,Z 102.535,A 171.717,B 90.000,C 0.000} C_DIS
LIN {X 287.019,Y -41.477,Z 102.492,A 171.777,B 90.000,C 0.000} C_DIS
LIN {X 287.028,Y -41.414,Z 102.441,A 171.790,B 90.000,C 0.000} C_DIS
LIN {X 287.034,Y -41.372,Z 102.390,A 171.798,B 90.000,C 0.000} C_DIS
LIN {X 287.063,Y -41.170,Z 102.348,A 171.838,B 90.000,C 0.000} C_DIS
LIN {X 287.069,Y -41.128,Z 102.297,A 171.847,B 90.000,C 0.000} C_DIS
LIN {X 287.078,Y -41.064,Z 102.246,A 171.859,B 90.000,C 0.000} C_DIS
LIN {X 287.121,Y -40.761,Z 102.203,A 171.920,B 90.000,C 0.000} C_DIS
LIN {X 287.139,Y -40.635,Z 102.101,A 171.945,B 90.000,C 0.000} C_DIS
LIN {X 287.182,Y -40.332,Z 102.059,A 172.006,B 90.000,C 0.000} C_DIS
LIN {X 287.199,Y -40.206,Z 101.957,A 172.031,B 90.000,C 0.000} C_DIS
LIN {X 287.242,Y -39.903,Z 101.914,A 172.091,B 90.000,C 0.000} C_DIS
LIN {X 287.250,Y -39.839,Z 101.863,A 172.104,B 90.000,C 0.000} C_DIS
LIN {X 287.256,Y -39.797,Z 101.812,A 172.112,B 90.000,C 0.000} C_DIS
LIN {X 287.284,Y -39.595,Z 101.770,A 172.153,B 90.000,C 0.000} C_DIS
LIN {X 287.290,Y -39.553,Z 101.719,A 172.161,B 90.000,C 0.000} C_DIS
LIN {X 287.299,Y -39.490,Z 101.668,A 172.174,B 90.000,C 0.000} C_DIS
LIN {X 287.340,Y -39.187,Z 101.625,A 172.234,B 90.000,C 0.000} C_DIS
LIN {X 287.357,Y -39.060,Z 101.523,A 172.259,B 90.000,C 0.000} C_DIS
LIN {X 287.398,Y -38.757,Z 101.481,A 172.320,B 90.000,C 0.000} C_DIS
LIN {X 287.415,Y -38.631,Z 101.378,A 172.345,B 90.000,C 0.000} C_DIS
LIN {X 287.456,Y -38.327,Z 101.336,A 172.405,B 90.000,C 0.000} C_DIS
LIN {X 287.465,Y -38.264,Z 101.285,A 172.418,B 90.000,C 0.000} C_DIS
LIN {X 287.470,Y -38.222,Z 101.234,A 172.426,B 90.000,C 0.000} C_DIS
LIN {X 287.497,Y -38.020,Z 101.191,A 172.467,B 90.000,C 0.000} C_DIS
LIN {X 287.503,Y -37.978,Z 101.140,A 172.475,B 90.000,C 0.000} C_DIS
LIN {X 287.511,Y -37.914,Z 101.089,A 172.488,B 90.000,C 0.000} C_DIS
LIN {X 287.551,Y -37.611,Z 101.047,A 172.548,B 90.000,C 0.000} C_DIS
LIN {X 287.567,Y -37.485,Z 100.945,A 172.573,B 90.000,C 0.000} C_DIS
LIN {X 287.607,Y -37.181,Z 100.902,A 172.634,B 90.000,C 0.000} C_DIS
LIN {X 287.623,Y -37.055,Z 100.800,A 172.659,B 90.000,C 0.000} C_DIS
LIN {X 287.662,Y -36.751,Z 100.758,A 172.719,B 90.000,C 0.000} C_DIS
LIN {X 287.670,Y -36.688,Z 100.707,A 172.732,B 90.000,C 0.000} C_DIS
LIN {X 287.675,Y -36.646,Z 100.656,A 172.740,B 90.000,C 0.000} C_DIS
LIN {X 287.701,Y -36.443,Z 100.613,A 172.781,B 90.000,C 0.000} C_DIS
LIN {X 287.706,Y -36.401,Z 100.562,A 172.789,B 90.000,C 0.000} C_DIS
LIN {X 287.714,Y -36.338,Z 100.511,A 172.802,B 90.000,C 0.000} C_DIS
LIN {X 287.753,Y -36.034,Z 100.469,A 172.862,B 90.000,C 0.000} C_DIS
LIN {X 287.768,Y -35.908,Z 100.367,A 172.887,B 90.000,C 0.000} C_DIS
LIN {X 287.806,Y -35.604,Z 100.324,A 172.948,B 90.000,C 0.000} C_DIS
LIN {X 287.814,Y -35.540,Z 100.273,A 172.961,B 90.000,C 0.000} C_DIS
LIN {X 287.819,Y -35.498,Z 100.222,A 172.969,B 90.000,C 0.000} C_DIS
LIN {X 287.844,Y -35.296,Z 100.180,A 173.009,B 90.000,C 0.000} C_DIS
LIN {X 287.854,Y -35.211,Z 100.078,A 173.026,B 90.000,C 0.000} C_DIS
LIN {X 287.880,Y -35.004,Z 100.045,A 173.067,B 90.000,C 0.000} C_DIS
LIN {X 287.883,Y -34.978,Z 100.001,A 173.072,B 90.000,C 0.000} C_DIS
LIN {X 287.839,Y -35.334,Z 99.595,A 173.002,B 90.000,C 0.000} C_DIS
LIN {X 287.826,Y -35.439,Z 99.364,A 172.981,B 90.000,C 0.000} C_DIS
LIN {X 287.801,Y -35.642,Z 99.150,A 172.940,B 90.000,C 0.000} C_DIS
LIN {X 287.796,Y -35.684,Z 99.029,A 172.932,B 90.000,C 0.000} C_DIS
LIN {X 287.794,Y -35.705,Z 98.938,A 172.928,B 90.000,C 0.000} C_DIS
LIN {X 287.781,Y -35.806,Z 98.858,A 172.908,B 90.000,C 0.000} C_DIS
LIN {X 287.776,Y -35.848,Z 98.654,A 172.899,B 90.000,C 0.000} C_DIS
LIN {X 287.763,Y -35.950,Z 98.569,A 172.879,B 90.000,C 0.000} C_DIS
LIN {X 287.758,Y -35.992,Z 98.365,A 172.871,B 90.000,C 0.000} C_DIS
LIN {X 287.752,Y -36.042,Z 98.322,A 172.861,B 90.000,C 0.000} C_DIS
LIN {X 287.745,Y -36.093,Z 98.258,A 172.850,B 90.000,C 0.000} C_DIS
LIN {X 287.740,Y -36.135,Z 97.952,A 172.842,B 90.000,C 0.000} C_DIS
LIN {X 287.734,Y -36.186,Z 97.889,A 172.832,B 90.000,C 0.000} C_DIS
LIN {X 287.727,Y -36.236,Z 97.804,A 172.822,B 90.000,C 0.000} C_DIS
LIN {X 287.722,Y -36.279,Z 97.395,A 172.814,B 90.000,C 0.000} C_DIS
LIN {X 287.715,Y -36.329,Z 97.310,A 172.803,B 90.000,C 0.000} C_DIS
LIN {X 287.709,Y -36.380,Z 97.166,A 172.793,B 90.000,C 0.000} C_DIS
LIN {X 287.704,Y -36.421,Z 96.443,A 172.785,B 90.000,C 0.000} C_DIS
LIN {X 287.697,Y -36.473,Z 96.299,A 172.775,B 90.000,C 0.000} C_DIS
LIN {X 287.691,Y -36.523,Z 96.214,A 172.765,B 90.000,C 0.000} C_DIS
LIN {X 287.688,Y -36.544,Z 96.010,A 172.761,B 90.000,C 0.000} C_DIS
LIN {X 287.691,Y -36.523,Z 95.806,A 172.765,B 90.000,C 0.000} C_DIS
LIN {X 287.697,Y -36.473,Z 95.721,A 172.775,B 90.000,C 0.000} C_DIS
LIN {X 287.704,Y -36.421,Z 95.558,A 172.785,B 90.000,C 0.000} C_DIS
LIN {X 287.709,Y -36.381,Z 94.727,A 172.793,B 90.000,C 0.000} C_DIS
LIN {X 287.715,Y -36.329,Z 94.564,A 172.803,B 90.000,C 0.000} C_DIS
LIN {X 287.722,Y -36.279,Z 94.479,A 172.814,B 90.000,C 0.000} C_DIS
LIN {X 287.727,Y -36.236,Z 94.071,A 172.822,B 90.000,C 0.000} C_DIS
LIN {X 287.734,Y -36.186,Z 93.986,A 172.832,B 90.000,C 0.000} C_DIS
LIN {X 287.740,Y -36.135,Z 93.944,A 172.842,B 90.000,C 0.000} C_DIS
LIN {X 287.745,Y -36.093,Z 93.740,A 172.850,B 90.000,C 0.000} C_DIS
LIN {X 287.752,Y -36.042,Z 93.697,A 172.861,B 90.000,C 0.000} C_DIS
LIN {X 287.758,Y -35.992,Z 93.638,A 172.871,B 90.000,C 0.000} C_DIS
LIN {X 287.766,Y -35.931,Z 93.323,A 172.883,B 90.000,C 0.000} C_DIS
LIN {X 287.791,Y -35.726,Z 93.080,A 172.924,B 90.000,C 0.000} C_DIS
LIN {X 287.796,Y -35.684,Z 92.959,A 172.932,B 90.000,C 0.000} C_DIS
LIN {X 287.799,Y -35.663,Z 92.868,A 172.936,B 90.000,C 0.000} C_DIS
LIN {X 287.811,Y -35.562,Z 92.792,A 172.956,B 90.000,C 0.000} C_DIS
LIN {X 287.814,Y -35.540,Z 92.701,A 172.961,B 90.000,C 0.000} C_DIS
LIN {X 287.819,Y -35.498,Z 92.580,A 172.969,B 90.000,C 0.000} C_DIS
LIN {X 287.832,Y -35.397,Z 92.469,A 172.989,B 90.000,C 0.000} C_DIS
LIN {X 287.869,Y -35.096,Z 92.046,A 173.049,B 90.000,C 0.000} C_DIS
LIN {X 287.963,Y -34.310,Z 91.255,A 173.205,B 90.000,C 0.000} C_DIS
LIN {X 288.013,Y -33.890,Z 90.951,A 173.289,B 90.000,C 0.000} C_DIS
LIN {X 288.025,Y -33.784,Z 90.849,A 173.310,B 90.000,C 0.000} C_DIS
LIN {X 288.051,Y -33.566,Z 90.764,A 173.353,B 90.000,C 0.000} C_DIS
LIN {X 288.076,Y -33.349,Z 90.560,A 173.397,B 90.000,C 0.000} C_DIS
LIN {X 288.090,Y -33.228,Z 90.518,A 173.421,B 90.000,C 0.000} C_DIS
LIN {X 288.100,Y -33.138,Z 90.496,A 173.438,B 90.000,C 0.000} C_DIS
LIN {X 288.110,Y -33.059,Z 90.394,A 173.454,B 90.000,C 0.000} C_DIS
LIN {X 288.133,Y -32.856,Z 90.352,A 173.495,B 90.000,C 0.000} C_DIS
LIN {X 288.138,Y -32.814,Z 90.301,A 173.503,B 90.000,C 0.000} C_DIS
LIN {X 288.145,Y -32.750,Z 90.250,A 173.516,B 90.000,C 0.000} C_DIS
LIN {X 288.179,Y -32.446,Z 90.207,A 173.576,B 90.000,C 0.000} C_DIS
LIN {X 288.193,Y -32.319,Z 90.105,A 173.601,B 90.000,C 0.000} C_DIS
LIN {X 288.227,Y -32.015,Z 90.063,A 173.662,B 90.000,C 0.000} C_DIS
LIN {X 288.234,Y -31.952,Z 90.012,A 173.674,B 90.000,C 0.000} C_DIS
LIN {X 288.244,Y -31.867,Z 89.961,A 173.691,B 90.000,C 0.000} C_DIS
LIN {X 288.288,Y -31.462,Z 89.918,A 173.772,B 90.000,C 0.000} C_DIS
LIN {X 288.298,Y -31.377,Z 89.867,A 173.789,B 90.000,C 0.000} C_DIS
LIN {X 288.327,Y -31.108,Z 89.814,A 173.842,B 90.000,C 0.000} C_DIS
LIN {X 288.482,Y -29.634,Z 89.814,A 174.135,B 90.000,C 0.000} C_DIS
LIN {X 288.509,Y -29.365,Z 89.867,A 174.188,B 90.000,C 0.000} C_DIS
LIN {X 288.520,Y -29.259,Z 89.918,A 174.209,B 90.000,C 0.000} C_DIS
LIN {X 288.571,Y -28.752,Z 89.961,A 174.310,B 90.000,C 0.000} C_DIS
LIN {X 288.582,Y -28.646,Z 90.012,A 174.331,B 90.000,C 0.000} C_DIS
LIN {X 288.588,Y -28.583,Z 90.063,A 174.344,B 90.000,C 0.000} C_DIS
LIN {X 288.618,Y -28.278,Z 90.105,A 174.404,B 90.000,C 0.000} C_DIS
LIN {X 288.630,Y -28.151,Z 90.207,A 174.429,B 90.000,C 0.000} C_DIS
LIN {X 288.660,Y -27.846,Z 90.250,A 174.490,B 90.000,C 0.000} C_DIS
LIN {X 288.666,Y -27.783,Z 90.301,A 174.502,B 90.000,C 0.000} C_DIS
LIN {X 288.670,Y -27.741,Z 90.352,A 174.511,B 90.000,C 0.000} C_DIS
LIN {X 288.690,Y -27.537,Z 90.394,A 174.551,B 90.000,C 0.000} C_DIS
LIN {X 288.697,Y -27.457,Z 90.496,A 174.567,B 90.000,C 0.000} C_DIS
LIN {X 288.706,Y -27.367,Z 90.518,A 174.585,B 90.000,C 0.000} C_DIS
LIN {X 288.717,Y -27.246,Z 90.560,A 174.609,B 90.000,C 0.000} C_DIS
LIN {X 288.737,Y -27.033,Z 90.764,A 174.651,B 90.000,C 0.000} C_DIS
LIN {X 288.759,Y -26.803,Z 90.870,A 174.697,B 90.000,C 0.000} C_DIS
LIN {X 288.843,Y -25.884,Z 91.591,A 174.879,B 90.000,C 0.000} C_DIS
LIN {X 288.859,Y -25.695,Z 91.668,A 174.917,B 90.000,C 0.000} C_DIS
LIN {X 288.873,Y -25.543,Z 91.676,A 174.947,B 90.000,C 0.000} C_DIS
LIN {X 288.878,Y -25.480,Z 91.602,A 174.959,B 90.000,C 0.000} C_DIS
LIN {X 288.886,Y -25.396,Z 91.551,A 174.976,B 90.000,C 0.000} C_DIS
LIN {X 288.921,Y -24.989,Z 91.508,A 175.057,B 90.000,C 0.000} C_DIS
LIN {X 288.929,Y -24.904,Z 91.457,A 175.074,B 90.000,C 0.000} C_DIS
LIN {X 288.934,Y -24.841,Z 91.406,A 175.086,B 90.000,C 0.000} C_DIS
LIN {X 288.960,Y -24.536,Z 91.364,A 175.147,B 90.000,C 0.000} C_DIS
LIN {X 288.966,Y -24.472,Z 91.313,A 175.159,B 90.000,C 0.000} C_DIS
LIN {X 288.973,Y -24.388,Z 91.261,A 175.176,B 90.000,C 0.000} C_DIS
LIN {X 289.007,Y -23.981,Z 91.219,A 175.257,B 90.000,C 0.000} C_DIS
LIN {X 289.014,Y -23.896,Z 91.168,A 175.273,B 90.000,C 0.000} C_DIS
LIN {X 289.019,Y -23.833,Z 91.117,A 175.286,B 90.000,C 0.000} C_DIS
LIN {X 289.044,Y -23.527,Z 91.074,A 175.347,B 90.000,C 0.000} C_DIS
LIN {X 289.049,Y -23.464,Z 91.023,A 175.359,B 90.000,C 0.000} C_DIS
LIN {X 289.056,Y -23.379,Z 90.972,A 175.376,B 90.000,C 0.000} C_DIS
LIN {X 289.089,Y -22.972,Z 90.930,A 175.457,B 90.000,C 0.000} C_DIS
LIN {X 289.095,Y -22.888,Z 90.879,A 175.473,B 90.000,C 0.000} C_DIS
LIN {X 289.100,Y -22.824,Z 90.828,A 175.486,B 90.000,C 0.000} C_DIS
LIN {X 289.124,Y -22.519,Z 90.785,A 175.546,B 90.000,C 0.000} C_DIS
LIN {X 289.134,Y -22.392,Z 90.683,A 175.572,B 90.000,C 0.000} C_DIS
LIN {X 289.158,Y -22.087,Z 90.641,A 175.632,B 90.000,C 0.000} C_DIS
LIN {X 289.163,Y -22.023,Z 90.590,A 175.645,B 90.000,C 0.000} C_DIS
LIN {X 289.180,Y -21.789,Z 90.537,A 175.691,B 90.000,C 0.000} C_DIS
LIN {X 289.273,Y -20.528,Z 90.537,A 175.941,B 90.000,C 0.000} C_DIS
LIN {X 289.289,Y -20.293,Z 90.590,A 175.987,B 90.000,C 0.000} C_DIS
LIN {X 289.293,Y -20.240,Z 90.641,A 175.998,B 90.000,C 0.000} C_DIS
LIN {X 289.302,Y -20.111,Z 90.662,A 176.023,B 90.000,C 0.000} C_DIS
LIN {X 289.317,Y -19.896,Z 90.754,A 176.066,B 90.000,C 0.000} C_DIS
LIN {X 289.335,Y -19.621,Z 90.971,A 176.120,B 90.000,C 0.000} C_DIS
LIN {X 289.351,Y -19.385,Z 91.222,A 176.167,B 90.000,C 0.000} C_DIS
LIN {X 289.358,Y -19.284,Z 91.419,A 176.187,B 90.000,C 0.000} C_DIS
LIN {X 289.360,Y -19.263,Z 91.497,A 176.191,B 90.000,C 0.000} C_DIS
LIN {X 289.363,Y -19.212,Z 91.529,A 176.201,B 90.000,C 0.000} C_DIS
LIN {X 289.366,Y -19.160,Z 91.692,A 176.212,B 90.000,C 0.000} C_DIS
LIN {X 289.366,Y -19.160,Z 92.523,A 176.212,B 90.000,C 0.000} C_DIS
LIN {X 289.363,Y -19.212,Z 92.686,A 176.201,B 90.000,C 0.000} C_DIS
LIN {X 289.360,Y -19.263,Z 92.745,A 176.191,B 90.000,C 0.000} C_DIS
LIN {X 289.355,Y -19.324,Z 93.060,A 176.179,B 90.000,C 0.000} C_DIS
LIN {X 289.339,Y -19.572,Z 93.390,A 176.130,B 90.000,C 0.000} C_DIS
LIN {X 289.334,Y -19.648,Z 93.536,A 176.115,B 90.000,C 0.000} C_DIS
LIN {X 289.322,Y -19.824,Z 93.735,A 176.080,B 90.000,C 0.000} C_DIS
LIN {X 289.308,Y -20.022,Z 93.911,A 176.041,B 90.000,C 0.000} C_DIS
LIN {X 289.298,Y -20.167,Z 93.986,A 176.012,B 90.000,C 0.000} C_DIS
LIN {X 289.284,Y -20.366,Z 94.131,A 175.973,B 90.000,C 0.000} C_DIS
LIN {X 289.276,Y -20.477,Z 94.233,A 175.951,B 90.000,C 0.000} C_DIS
LIN {X 289.268,Y -20.598,Z 94.275,A 175.927,B 90.000,C 0.000} C_DIS
LIN {X 289.261,Y -20.688,Z 94.297,A 175.909,B 90.000,C 0.000} C_DIS
LIN {X 289.255,Y -20.768,Z 94.399,A 175.893,B 90.000,C 0.000} C_DIS
LIN {X 289.241,Y -20.972,Z 94.441,A 175.853,B 90.000,C 0.000} C_DIS
LIN {X 289.235,Y -21.057,Z 94.543,A 175.836,B 90.000,C 0.000} C_DIS
LIN {X 289.220,Y -21.260,Z 94.586,A 175.796,B 90.000,C 0.000} C_DIS
LIN {X 289.213,Y -21.345,Z 94.688,A 175.779,B 90.000,C 0.000} C_DIS
LIN {X 289.198,Y -21.548,Z 94.730,A 175.739,B 90.000,C 0.000} C_DIS
LIN {X 289.195,Y -21.591,Z 94.781,A 175.730,B 90.000,C 0.000} C_DIS
LIN {X 289.190,Y -21.654,Z 94.832,A 175.718,B 90.000,C 0.000} C_DIS
LIN {X 289.167,Y -21.960,Z 94.875,A 175.657,B 90.000,C 0.000} C_DIS
LIN {X 289.163,Y -22.023,Z 94.926,A 175.645,B 90.000,C 0.000} C_DIS
LIN {X 289.159,Y -22.065,Z 94.977,A 175.636,B 90.000,C 0.000} C_DIS
LIN {X 289.144,Y -22.269,Z 95.019,A 175.596,B 90.000,C 0.000} C_DIS
LIN {X 289.137,Y -22.354,Z 95.121,A 175.579,B 90.000,C 0.000} C_DIS
LIN {X 289.121,Y -22.557,Z 95.164,A 175.539,B 90.000,C 0.000} C_DIS
LIN {X 289.115,Y -22.642,Z 95.266,A 175.522,B 90.000,C 0.000} C_DIS
LIN {X 289.099,Y -22.845,Z 95.308,A 175.482,B 90.000,C 0.000} C_DIS
LIN {X 289.092,Y -22.930,Z 95.410,A 175.465,B 90.000,C 0.000} C_DIS
LIN {X 289.076,Y -23.134,Z 95.453,A 175.425,B 90.000,C 0.000} C_DIS
LIN {X 289.069,Y -23.218,Z 95.555,A 175.408,B 90.000,C 0.000} C_DIS
LIN {X 289.053,Y -23.422,Z 95.597,A 175.368,B 90.000,C 0.000} C_DIS
LIN {X 289.046,Y -23.506,Z 95.699,A 175.351,B 90.000,C 0.000} C_DIS
LIN {X 289.029,Y -23.710,Z 95.742,A 175.310,B 90.000,C 0.000} C_DIS
LIN {X 289.022,Y -23.794,Z 95.844,A 175.294,B 90.000,C 0.000} C_DIS
LIN {X 289.005,Y -23.998,Z 95.886,A 175.253,B 90.000,C 0.000} C_DIS
LIN {X 289.002,Y -24.040,Z 95.937,A 175.245,B 90.000,C 0.000} C_DIS
LIN {X 289.005,Y -23.998,Z 95.989,A 175.253,B 90.000,C 0.000} C_DIS
LIN {X 289.014,Y -23.896,Z 96.010,A 175.273,B 90.000,C 0.000} C_DIS
LIN {X 289.022,Y -23.794,Z 95.989,A 175.294,B 90.000,C 0.000} C_DIS
LIN {X 289.026,Y -23.752,Z 95.937,A 175.302,B 90.000,C 0.000} C_DIS
LIN {X 289.031,Y -23.689,Z 95.886,A 175.315,B 90.000,C 0.000} C_DIS
LIN {X 289.056,Y -23.383,Z 95.844,A 175.375,B 90.000,C 0.000} C_DIS
LIN {X 289.061,Y -23.320,Z 95.793,A 175.388,B 90.000,C 0.000} C_DIS
LIN {X 289.064,Y -23.278,Z 95.742,A 175.396,B 90.000,C 0.000} C_DIS
LIN {X 289.081,Y -23.074,Z 95.699,A 175.436,B 90.000,C 0.000} C_DIS
LIN {X 289.084,Y -23.032,Z 95.648,A 175.445,B 90.000,C 0.000} C_DIS
LIN {X 289.089,Y -22.968,Z 95.597,A 175.457,B 90.000,C 0.000} C_DIS
LIN {X 289.113,Y -22.663,Z 95.555,A 175.518,B 90.000,C 0.000} C_DIS
LIN {X 289.118,Y -22.600,Z 95.504,A 175.530,B 90.000,C 0.000} C_DIS
LIN {X 289.125,Y -22.515,Z 95.453,A 175.547,B 90.000,C 0.000} C_DIS
LIN {X 289.140,Y -22.311,Z 95.432,A 175.588,B 90.000,C 0.000} C_DIS
LIN {X 289.156,Y -22.108,Z 95.453,A 175.628,B 90.000,C 0.000} C_DIS
LIN {X 289.163,Y -22.023,Z 95.504,A 175.645,B 90.000,C 0.000} C_DIS
LIN {X 289.165,Y -21.990,Z 95.555,A 175.651,B 90.000,C 0.000} C_DIS
LIN {X 289.180,Y -21.799,Z 95.606,A 175.689,B 90.000,C 0.000} C_DIS
LIN {X 289.187,Y -21.696,Z 95.681,A 175.710,B 90.000,C 0.000} C_DIS
LIN {X 289.193,Y -21.620,Z 95.785,A 175.725,B 90.000,C 0.000} C_DIS
LIN {X 289.197,Y -21.570,Z 95.976,A 175.735,B 90.000,C 0.000} C_DIS
LIN {X 289.201,Y -21.519,Z 96.010,A 175.745,B 90.000,C 0.000} C_DIS
LIN {X 289.204,Y -21.466,Z 96.353,A 175.755,B 90.000,C 0.000} C_DIS
LIN {X 289.207,Y -21.428,Z 98.268,A 175.763,B 90.000,C 0.000} C_DIS
LIN {X 289.215,Y -21.321,Z 99.055,A 175.784,B 90.000,C 0.000} C_DIS
LIN {X 289.217,Y -21.302,Z 101.555,A 175.787,B 90.000,C 0.000} C_DIS
LIN {X 289.217,Y -21.302,Z 102.014,A 175.787,B 90.000,C 0.000} C_DIS
LIN {X 289.203,Y -21.479,Z 102.192,A 175.752,B 90.000,C 0.000} C_DIS
LIN {X 289.192,Y -21.637,Z 102.317,A 175.721,B 90.000,C 0.000} C_DIS
LIN {X 289.182,Y -21.768,Z 102.369,A 175.695,B 90.000,C 0.000} C_DIS
LIN {X 289.176,Y -21.846,Z 102.390,A 175.680,B 90.000,C 0.000} C_DIS
LIN {X 289.173,Y -21.879,Z 102.441,A 175.673,B 90.000,C 0.000} C_DIS
LIN {X 289.170,Y -21.921,Z 102.492,A 175.665,B 90.000,C 0.000} C_DIS
LIN {X 289.155,Y -22.125,Z 102.535,A 175.625,B 90.000,C 0.000} C_DIS
LIN {X 289.148,Y -22.209,Z 102.637,A 175.608,B 90.000,C 0.000} C_DIS
LIN {X 289.133,Y -22.413,Z 102.679,A 175.567,B 90.000,C 0.000} C_DIS
LIN {X 289.129,Y -22.455,Z 102.730,A 175.559,B 90.000,C 0.000} C_DIS
LIN {X 289.124,Y -22.519,Z 102.781,A 175.546,B 90.000,C 0.000} C_DIS
LIN {X 289.100,Y -22.824,Z 102.824,A 175.486,B 90.000,C 0.000} C_DIS
LIN {X 289.095,Y -22.888,Z 102.875,A 175.473,B 90.000,C 0.000} C_DIS
LIN {X 289.092,Y -22.930,Z 102.926,A 175.465,B 90.000,C 0.000} C_DIS
LIN {X 289.076,Y -23.133,Z 102.968,A 175.425,B 90.000,C 0.000} C_DIS
LIN {X 289.072,Y -23.176,Z 103.019,A 175.416,B 90.000,C 0.000} C_DIS
LIN {X 289.067,Y -23.239,Z 103.070,A 175.404,B 90.000,C 0.000} C_DIS
LIN {X 289.043,Y -23.544,Z 103.113,A 175.343,B 90.000,C 0.000} C_DIS
LIN {X 289.037,Y -23.608,Z 103.164,A 175.331,B 90.000,C 0.000} C_DIS
LIN {X 289.034,Y -23.650,Z 103.215,A 175.322,B 90.000,C 0.000} C_DIS
LIN {X 289.017,Y -23.854,Z 103.257,A 175.282,B 90.000,C 0.000} C_DIS
LIN {X 289.010,Y -23.938,Z 103.359,A 175.265,B 90.000,C 0.000} C_DIS
LIN {X 288.993,Y -24.142,Z 103.402,A 175.225,B 90.000,C 0.000} C_DIS
LIN {X 288.986,Y -24.226,Z 103.504,A 175.208,B 90.000,C 0.000} C_DIS
LIN {X 288.969,Y -24.430,Z 103.546,A 175.168,B 90.000,C 0.000} C_DIS
LIN {X 288.966,Y -24.472,Z 103.597,A 175.159,B 90.000,C 0.000} C_DIS
LIN {X 288.960,Y -24.536,Z 103.649,A 175.147,B 90.000,C 0.000} C_DIS
LIN {X 288.934,Y -24.841,Z 103.691,A 175.086,B 90.000,C 0.000} C_DIS
LIN {X 288.929,Y -24.904,Z 103.742,A 175.074,B 90.000,C 0.000} C_DIS
LIN {X 288.925,Y -24.946,Z 103.793,A 175.065,B 90.000,C 0.000} C_DIS
LIN {X 288.907,Y -25.150,Z 103.835,A 175.025,B 90.000,C 0.000} C_DIS
LIN {X 288.904,Y -25.192,Z 103.887,A 175.016,B 90.000,C 0.000} C_DIS
LIN {X 288.898,Y -25.256,Z 103.938,A 175.004,B 90.000,C 0.000} C_DIS
LIN {X 288.871,Y -25.561,Z 103.980,A 174.943,B 90.000,C 0.000} C_DIS
LIN {X 288.866,Y -25.624,Z 104.031,A 174.931,B 90.000,C 0.000} C_DIS
LIN {X 288.862,Y -25.666,Z 104.082,A 174.922,B 90.000,C 0.000} C_DIS
LIN {X 288.844,Y -25.870,Z 104.125,A 174.882,B 90.000,C 0.000} C_DIS
LIN {X 288.836,Y -25.954,Z 104.227,A 174.865,B 90.000,C 0.000} C_DIS
LIN {X 288.818,Y -26.158,Z 104.269,A 174.825,B 90.000,C 0.000} C_DIS
LIN {X 288.814,Y -26.200,Z 104.320,A 174.817,B 90.000,C 0.000} C_DIS
LIN {X 288.808,Y -26.263,Z 104.371,A 174.804,B 90.000,C 0.000} C_DIS
LIN {X 288.780,Y -26.568,Z 104.414,A 174.744,B 90.000,C 0.000} C_DIS
LIN {X 288.775,Y -26.632,Z 104.465,A 174.731,B 90.000,C 0.000} C_DIS
LIN {X 288.771,Y -26.674,Z 104.516,A 174.723,B 90.000,C 0.000} C_DIS
LIN {X 288.752,Y -26.877,Z 104.558,A 174.682,B 90.000,C 0.000} C_DIS
LIN {X 288.744,Y -26.962,Z 104.660,A 174.665,B 90.000,C 0.000} C_DIS
LIN {X 288.725,Y -27.165,Z 104.703,A 174.625,B 90.000,C 0.000} C_DIS
LIN {X 288.721,Y -27.207,Z 104.754,A 174.617,B 90.000,C 0.000} C_DIS
LIN {X 288.715,Y -27.271,Z 104.805,A 174.604,B 90.000,C 0.000} C_DIS
LIN {X 288.686,Y -27.575,Z 104.847,A 174.544,B 90.000,C 0.000} C_DIS
LIN {X 288.680,Y -27.639,Z 104.898,A 174.531,B 90.000,C 0.000} C_DIS
LIN {X 288.676,Y -27.681,Z 104.949,A 174.523,B 90.000,C 0.000} C_DIS
LIN {X 288.656,Y -27.884,Z 104.992,A 174.482,B 90.000,C 0.000} C_DIS
LIN {X 288.648,Y -27.969,Z 105.094,A 174.466,B 90.000,C 0.000} C_DIS
LIN {X 288.628,Y -28.172,Z 105.136,A 174.425,B 90.000,C 0.000} C_DIS
LIN {X 288.624,Y -28.214,Z 105.187,A 174.417,B 90.000,C 0.000} C_DIS
LIN {X 288.618,Y -28.278,Z 105.238,A 174.404,B 90.000,C 0.000} C_DIS
LIN {X 288.588,Y -28.582,Z 105.281,A 174.344,B 90.000,C 0.000} C_DIS
LIN {X 288.582,Y -28.646,Z 105.332,A 174.331,B 90.000,C 0.000} C_DIS
LIN {X 288.578,Y -28.688,Z 105.383,A 174.323,B 90.000,C 0.000} C_DIS
LIN {X 288.557,Y -28.891,Z 105.425,A 174.282,B 90.000,C 0.000} C_DIS
LIN {X 288.553,Y -28.933,Z 105.476,A 174.274,B 90.000,C 0.000} C_DIS
LIN {X 288.547,Y -28.997,Z 105.527,A 174.261,B 90.000,C 0.000} C_DIS
LIN {X 288.516,Y -29.301,Z 105.570,A 174.201,B 90.000,C 0.000} C_DIS
LIN {X 288.509,Y -29.365,Z 105.621,A 174.188,B 90.000,C 0.000} C_DIS
LIN {X 288.505,Y -29.407,Z 105.672,A 174.180,B 90.000,C 0.000} C_DIS
LIN {X 288.484,Y -29.610,Z 105.714,A 174.140,B 90.000,C 0.000} C_DIS
LIN {X 288.476,Y -29.695,Z 105.816,A 174.123,B 90.000,C 0.000} C_DIS
LIN {X 288.455,Y -29.898,Z 105.859,A 174.083,B 90.000,C 0.000} C_DIS
LIN {X 288.450,Y -29.940,Z 105.910,A 174.074,B 90.000,C 0.000} C_DIS
LIN {X 288.444,Y -30.003,Z 105.961,A 174.062,B 90.000,C 0.000} C_DIS
LIN {X 288.412,Y -30.308,Z 106.003,A 174.001,B 90.000,C 0.000} C_DIS
LIN {X 288.405,Y -30.371,Z 106.054,A 173.989,B 90.000,C 0.000} C_DIS
LIN {X 288.401,Y -30.413,Z 106.105,A 173.980,B 90.000,C 0.000} C_DIS
LIN {X 288.379,Y -30.616,Z 106.148,A 173.940,B 90.000,C 0.000} C_DIS
LIN {X 288.370,Y -30.701,Z 106.250,A 173.923,B 90.000,C 0.000} C_DIS
LIN {X 288.349,Y -30.904,Z 106.292,A 173.883,B 90.000,C 0.000} C_DIS
LIN {X 288.344,Y -30.946,Z 106.344,A 173.874,B 90.000,C 0.000} C_DIS
LIN {X 288.337,Y -31.009,Z 106.395,A 173.862,B 90.000,C 0.000} C_DIS
LIN {X 288.304,Y -31.314,Z 106.437,A 173.801,B 90.000,C 0.000} C_DIS
LIN {X 288.298,Y -31.377,Z 106.488,A 173.789,B 90.000,C 0.000} C_DIS
LIN {X 288.293,Y -31.419,Z 106.539,A 173.780,B 90.000,C 0.000} C_DIS
LIN {X 288.271,Y -31.622,Z 106.582,A 173.740,B 90.000,C 0.000} C_DIS
LIN {X 288.261,Y -31.707,Z 106.684,A 173.723,B 90.000,C 0.000} C_DIS
LIN {X 288.239,Y -31.910,Z 106.726,A 173.683,B 90.000,C 0.000} C_DIS
LIN {X 288.234,Y -31.952,Z 106.777,A 173.674,B 90.000,C 0.000} C_DIS
LIN {X 288.227,Y -32.015,Z 106.828,A 173.662,B 90.000,C 0.000} C_DIS
LIN {X 288.193,Y -32.319,Z 106.871,A 173.601,B 90.000,C 0.000} C_DIS
LIN {X 288.186,Y -32.383,Z 106.922,A 173.589,B 90.000,C 0.000} C_DIS
LIN {X 288.182,Y -32.425,Z 106.973,A 173.580,B 90.000,C 0.000} C_DIS
LIN {X 288.159,Y -32.628,Z 107.015,A 173.540,B 90.000,C 0.000} C_DIS
LIN {X 288.154,Y -32.670,Z 107.066,A 173.532,B 90.000,C 0.000} C_DIS
LIN {X 288.147,Y -32.733,Z 107.117,A 173.519,B 90.000,C 0.000} C_DIS
LIN {X 288.112,Y -33.037,Z 107.160,A 173.459,B 90.000,C 0.000} C_DIS
LIN {X 288.105,Y -33.101,Z 107.211,A 173.446,B 90.000,C 0.000} C_DIS
LIN {X 288.100,Y -33.143,Z 107.262,A 173.438,B 90.000,C 0.000} C_DIS
LIN {X 288.076,Y -33.346,Z 107.304,A 173.397,B 90.000,C 0.000} C_DIS
LIN {X 288.067,Y -33.430,Z 107.406,A 173.380,B 90.000,C 0.000} C_DIS
LIN {X 288.043,Y -33.633,Z 107.449,A 173.340,B 90.000,C 0.000} C_DIS
LIN {X 288.038,Y -33.675,Z 107.500,A 173.332,B 90.000,C 0.000} C_DIS
LIN {X 288.031,Y -33.738,Z 107.551,A 173.319,B 90.000,C 0.000} C_DIS
LIN {X 287.995,Y -34.042,Z 107.593,A 173.259,B 90.000,C 0.000} C_DIS
LIN {X 287.988,Y -34.106,Z 107.644,A 173.246,B 90.000,C 0.000} C_DIS
LIN {X 287.983,Y -34.148,Z 107.695,A 173.238,B 90.000,C 0.000} C_DIS
LIN {X 287.958,Y -34.350,Z 107.738,A 173.197,B 90.000,C 0.000} C_DIS
LIN {X 287.948,Y -34.435,Z 107.840,A 173.181,B 90.000,C 0.000} C_DIS
LIN {X 287.924,Y -34.637,Z 107.882,A 173.140,B 90.000,C 0.000} C_DIS
LIN {X 287.919,Y -34.680,Z 107.933,A 173.132,B 90.000,C 0.000} C_DIS
LIN {X 287.911,Y -34.743,Z 107.984,A 173.119,B 90.000,C 0.000} C_DIS
LIN {X 287.874,Y -35.047,Z 108.027,A 173.059,B 90.000,C 0.000} C_DIS
LIN {X 287.867,Y -35.110,Z 108.078,A 173.046,B 90.000,C 0.000} C_DIS
LIN {X 287.862,Y -35.152,Z 108.129,A 173.038,B 90.000,C 0.000} C_DIS
LIN {X 287.837,Y -35.355,Z 108.171,A 172.997,B 90.000,C 0.000} C_DIS
LIN {X 287.826,Y -35.439,Z 108.273,A 172.981,B 90.000,C 0.000} C_DIS
LIN {X 287.801,Y -35.642,Z 108.316,A 172.940,B 90.000,C 0.000} C_DIS
LIN {X 287.796,Y -35.684,Z 108.367,A 172.932,B 90.000,C 0.000} C_DIS
LIN {X 287.788,Y -35.747,Z 108.418,A 172.919,B 90.000,C 0.000} C_DIS
LIN {X 287.750,Y -36.051,Z 108.460,A 172.859,B 90.000,C 0.000} C_DIS
LIN {X 287.743,Y -36.114,Z 108.511,A 172.846,B 90.000,C 0.000} C_DIS
LIN {X 287.737,Y -36.156,Z 108.562,A 172.838,B 90.000,C 0.000} C_DIS
LIN {X 287.712,Y -36.359,Z 108.605,A 172.798,B 90.000,C 0.000} C_DIS
LIN {X 287.706,Y -36.401,Z 108.656,A 172.789,B 90.000,C 0.000} C_DIS
LIN {X 287.698,Y -36.464,Z 108.707,A 172.777,B 90.000,C 0.000} C_DIS
LIN {X 287.660,Y -36.768,Z 108.749,A 172.716,B 90.000,C 0.000} C_DIS
LIN {X 287.652,Y -36.831,Z 108.800,A 172.704,B 90.000,C 0.000} C_DIS
LIN {X 287.646,Y -36.873,Z 108.852,A 172.695,B 90.000,C 0.000} C_DIS
LIN {X 287.620,Y -37.076,Z 108.894,A 172.655,B 90.000,C 0.000} C_DIS
LIN {X 287.609,Y -37.160,Z 108.996,A 172.638,B 90.000,C 0.000} C_DIS
LIN {X 287.583,Y -37.362,Z 109.039,A 172.598,B 90.000,C 0.000} C_DIS
LIN {X 287.578,Y -37.404,Z 109.090,A 172.589,B 90.000,C 0.000} C_DIS
LIN {X 287.569,Y -37.467,Z 109.141,A 172.577,B 90.000,C 0.000} C_DIS
LIN {X 287.530,Y -37.771,Z 109.183,A 172.516,B 90.000,C 0.000} C_DIS
LIN {X 287.521,Y -37.834,Z 109.234,A 172.504,B 90.000,C 0.000} C_DIS
LIN {X 287.516,Y -37.876,Z 109.285,A 172.495,B 90.000,C 0.000} C_DIS
LIN {X 287.489,Y -38.079,Z 109.328,A 172.455,B 90.000,C 0.000} C_DIS
LIN {X 287.478,Y -38.163,Z 109.430,A 172.438,B 90.000,C 0.000} C_DIS
LIN {X 287.451,Y -38.365,Z 109.472,A 172.398,B 90.000,C 0.000} C_DIS
LIN {X 287.445,Y -38.407,Z 109.523,A 172.389,B 90.000,C 0.000} C_DIS
LIN {X 287.437,Y -38.470,Z 109.574,A 172.377,B 90.000,C 0.000} C_DIS
LIN {X 287.396,Y -38.774,Z 109.617,A 172.316,B 90.000,C 0.000} C_DIS
LIN {X 287.388,Y -38.837,Z 109.668,A 172.304,B 90.000,C 0.000} C_DIS
LIN {X 287.382,Y -38.879,Z 109.719,A 172.295,B 90.000,C 0.000} C_DIS
LIN {X 287.355,Y -39.081,Z 109.761,A 172.255,B 90.000,C 0.000} C_DIS
LIN {X 287.343,Y -39.166,Z 109.863,A 172.238,B 90.000,C 0.000} C_DIS
LIN {X 287.315,Y -39.368,Z 109.906,A 172.198,B 90.000,C 0.000} C_DIS
LIN {X 287.310,Y -39.410,Z 109.957,A 172.190,B 90.000,C 0.000} C_DIS
LIN {X 287.301,Y -39.473,Z 110.008,A 172.177,B 90.000,C 0.000} C_DIS
LIN {X 287.259,Y -39.776,Z 110.050,A 172.116,B 90.000,C 0.000} C_DIS
LIN {X 287.250,Y -39.839,Z 110.101,A 172.104,B 90.000,C 0.000} C_DIS
LIN {X 287.245,Y -39.881,Z 110.152,A 172.096,B 90.000,C 0.000} C_DIS
LIN {X 287.216,Y -40.084,Z 110.195,A 172.055,B 90.000,C 0.000} C_DIS
LIN {X 287.205,Y -40.168,Z 110.297,A 172.038,B 90.000,C 0.000} C_DIS
LIN {X 287.176,Y -40.370,Z 110.339,A 171.998,B 90.000,C 0.000} C_DIS
LIN {X 287.170,Y -40.412,Z 110.390,A 171.990,B 90.000,C 0.000} C_DIS
LIN {X 287.162,Y -40.475,Z 110.441,A 171.977,B 90.000,C 0.000} C_DIS
LIN {X 287.119,Y -40.778,Z 110.484,A 171.917,B 90.000,C 0.000} C_DIS
LIN {X 287.110,Y -40.841,Z 110.535,A 171.904,B 90.000,C 0.000} C_DIS
LIN {X 287.104,Y -40.883,Z 110.586,A 171.896,B 90.000,C 0.000} C_DIS
LIN {X 287.075,Y -41.085,Z 110.628,A 171.855,B 90.000,C 0.000} C_DIS
LIN {X 287.069,Y -41.127,Z 110.679,A 171.847,B 90.000,C 0.000} C_DIS
LIN {X 287.060,Y -41.190,Z 110.730,A 171.834,B 90.000,C 0.000} C_DIS
LIN {X 287.016,Y -41.494,Z 110.773,A 171.774,B 90.000,C 0.000} C_DIS
LIN {X 287.007,Y -41.557,Z 110.824,A 171.761,B 90.000,C 0.000} C_DIS
LIN {X 287.001,Y -41.599,Z 110.875,A 171.753,B 90.000,C 0.000} C_DIS
LIN {X 286.972,Y -41.801,Z 110.917,A 171.713,B 90.000,C 0.000} C_DIS
LIN {X 286.959,Y -41.885,Z 111.019,A 171.696,B 90.000,C 0.000} C_DIS
LIN {X 286.930,Y -42.087,Z 111.062,A 171.655,B 90.000,C 0.000} C_DIS
LIN {X 286.924,Y -42.129,Z 111.113,A 171.647,B 90.000,C 0.000} C_DIS
LIN {X 286.914,Y -42.192,Z 111.164,A 171.634,B 90.000,C 0.000} C_DIS
LIN {X 286.870,Y -42.495,Z 111.206,A 171.574,B 90.000,C 0.000} C_DIS
LIN {X 286.860,Y -42.558,Z 111.257,A 171.561,B 90.000,C 0.000} C_DIS
LIN {X 286.854,Y -42.600,Z 111.308,A 171.553,B 90.000,C 0.000} C_DIS
LIN {X 286.824,Y -42.801,Z 111.351,A 171.513,B 90.000,C 0.000} C_DIS
LIN {X 286.812,Y -42.885,Z 111.453,A 171.496,B 90.000,C 0.000} C_DIS
LIN {X 286.781,Y -43.087,Z 111.495,A 171.456,B 90.000,C 0.000} C_DIS
LIN {X 286.775,Y -43.129,Z 111.547,A 171.447,B 90.000,C 0.000} C_DIS
LIN {X 286.765,Y -43.192,Z 111.598,A 171.435,B 90.000,C 0.000} C_DIS
LIN {X 286.720,Y -43.495,Z 111.640,A 171.374,B 90.000,C 0.000} C_DIS
LIN {X 286.710,Y -43.558,Z 111.691,A 171.361,B 90.000,C 0.000} C_DIS
LIN {X 286.704,Y -43.600,Z 111.742,A 171.353,B 90.000,C 0.000} C_DIS
LIN {X 286.673,Y -43.802,Z 111.785,A 171.313,B 90.000,C 0.000} C_DIS
LIN {X 286.660,Y -43.886,Z 111.887,A 171.296,B 90.000,C 0.000} C_DIS
LIN {X 286.629,Y -44.088,Z 111.929,A 171.256,B 90.000,C 0.000} C_DIS
LIN {X 286.623,Y -44.130,Z 111.980,A 171.247,B 90.000,C 0.000} C_DIS
LIN {X 286.613,Y -44.192,Z 112.031,A 171.235,B 90.000,C 0.000} C_DIS
LIN {X 286.566,Y -44.495,Z 112.074,A 171.174,B 90.000,C 0.000} C_DIS
LIN {X 286.556,Y -44.558,Z 112.125,A 171.162,B 90.000,C 0.000} C_DIS
LIN {X 286.550,Y -44.600,Z 112.176,A 171.153,B 90.000,C 0.000} C_DIS
LIN {X 286.518,Y -44.802,Z 112.218,A 171.113,B 90.000,C 0.000} C_DIS
LIN {X 286.505,Y -44.886,Z 112.320,A 171.096,B 90.000,C 0.000} C_DIS
LIN {X 286.474,Y -45.087,Z 112.363,A 171.056,B 90.000,C 0.000} C_DIS
LIN {X 286.467,Y -45.129,Z 112.414,A 171.047,B 90.000,C 0.000} C_DIS
LIN {X 286.457,Y -45.192,Z 112.465,A 171.035,B 90.000,C 0.000} C_DIS
LIN {X 286.409,Y -45.495,Z 112.507,A 170.974,B 90.000,C 0.000} C_DIS
LIN {X 286.399,Y -45.557,Z 112.558,A 170.962,B 90.000,C 0.000} C_DIS
LIN {X 286.393,Y -45.599,Z 112.609,A 170.953,B 90.000,C 0.000} C_DIS
LIN {X 286.360,Y -45.801,Z 112.652,A 170.913,B 90.000,C 0.000} C_DIS
LIN {X 286.354,Y -45.843,Z 112.703,A 170.905,B 90.000,C 0.000} C_DIS
LIN {X 286.344,Y -45.906,Z 112.754,A 170.892,B 90.000,C 0.000} C_DIS
LIN {X 286.295,Y -46.208,Z 112.796,A 170.832,B 90.000,C 0.000} C_DIS
LIN {X 286.285,Y -46.271,Z 112.847,A 170.819,B 90.000,C 0.000} C_DIS
LIN {X 286.278,Y -46.313,Z 112.898,A 170.811,B 90.000,C 0.000} C_DIS
LIN {X 286.245,Y -46.514,Z 112.941,A 170.770,B 90.000,C 0.000} C_DIS
LIN {X 286.232,Y -46.598,Z 113.043,A 170.753,B 90.000,C 0.000} C_DIS
LIN {X 286.199,Y -46.800,Z 113.085,A 170.713,B 90.000,C 0.000} C_DIS
LIN {X 286.192,Y -46.842,Z 113.136,A 170.705,B 90.000,C 0.000} C_DIS
LIN {X 286.182,Y -46.904,Z 113.187,A 170.692,B 90.000,C 0.000} C_DIS
LIN {X 286.132,Y -47.207,Z 113.230,A 170.632,B 90.000,C 0.000} C_DIS
LIN {X 286.122,Y -47.269,Z 113.281,A 170.619,B 90.000,C 0.000} C_DIS
LIN {X 286.115,Y -47.311,Z 113.332,A 170.611,B 90.000,C 0.000} C_DIS
LIN {X 286.081,Y -47.513,Z 113.374,A 170.570,B 90.000,C 0.000} C_DIS
LIN {X 286.067,Y -47.596,Z 113.476,A 170.554,B 90.000,C 0.000} C_DIS
LIN {X 286.034,Y -47.798,Z 113.519,A 170.513,B 90.000,C 0.000} C_DIS
LIN {X 286.027,Y -47.840,Z 113.570,A 170.505,B 90.000,C 0.000} C_DIS
LIN {X 286.016,Y -47.902,Z 113.621,A 170.492,B 90.000,C 0.000} C_DIS
LIN {X 285.966,Y -48.204,Z 113.663,A 170.432,B 90.000,C 0.000} C_DIS
LIN {X 285.955,Y -48.267,Z 113.714,A 170.419,B 90.000,C 0.000} C_DIS
LIN {X 285.948,Y -48.309,Z 113.765,A 170.411,B 90.000,C 0.000} C_DIS
LIN {X 285.914,Y -48.510,Z 113.808,A 170.370,B 90.000,C 0.000} C_DIS
LIN {X 285.900,Y -48.594,Z 113.910,A 170.354,B 90.000,C 0.000} C_DIS
LIN {X 285.865,Y -48.795,Z 113.952,A 170.313,B 90.000,C 0.000} C_DIS
LIN {X 285.858,Y -48.837,Z 114.003,A 170.305,B 90.000,C 0.000} C_DIS
LIN {X 285.847,Y -48.900,Z 114.055,A 170.292,B 90.000,C 0.000} C_DIS
LIN {X 285.796,Y -49.202,Z 114.097,A 170.232,B 90.000,C 0.000} C_DIS
LIN {X 285.785,Y -49.265,Z 114.148,A 170.219,B 90.000,C 0.000} C_DIS
LIN {X 285.778,Y -49.306,Z 114.199,A 170.211,B 90.000,C 0.000} C_DIS
LIN {X 285.743,Y -49.508,Z 114.242,A 170.171,B 90.000,C 0.000} C_DIS
LIN {X 285.736,Y -49.549,Z 114.293,A 170.162,B 90.000,C 0.000} C_DIS
LIN {X 285.725,Y -49.612,Z 114.344,A 170.150,B 90.000,C 0.000} C_DIS
LIN {X 285.672,Y -49.914,Z 114.386,A 170.089,B 90.000,C 0.000} C_DIS
LIN {X 285.661,Y -49.977,Z 114.437,A 170.077,B 90.000,C 0.000} C_DIS
LIN {X 285.654,Y -50.018,Z 114.488,A 170.068,B 90.000,C 0.000} C_DIS
LIN {X 285.619,Y -50.219,Z 114.531,A 170.028,B 90.000,C 0.000} C_DIS
LIN {X 285.604,Y -50.303,Z 114.633,A 170.011,B 90.000,C 0.000} C_DIS
LIN {X 285.568,Y -50.504,Z 114.675,A 169.971,B 90.000,C 0.000} C_DIS
LIN {X 285.561,Y -50.546,Z 114.726,A 169.962,B 90.000,C 0.000} C_DIS
LIN {X 285.550,Y -50.609,Z 114.777,A 169.950,B 90.000,C 0.000} C_DIS
LIN {X 285.496,Y -50.910,Z 114.820,A 169.889,B 90.000,C 0.000} C_DIS
LIN {X 285.485,Y -50.973,Z 114.871,A 169.877,B 90.000,C 0.000} C_DIS
LIN {X 285.478,Y -51.015,Z 114.922,A 169.868,B 90.000,C 0.000} C_DIS
LIN {X 285.442,Y -51.216,Z 114.964,A 169.828,B 90.000,C 0.000} C_DIS
LIN {X 285.427,Y -51.299,Z 115.066,A 169.811,B 90.000,C 0.000} C_DIS
LIN {X 285.391,Y -51.500,Z 115.109,A 169.771,B 90.000,C 0.000} C_DIS
LIN {X 285.383,Y -51.542,Z 115.160,A 169.762,B 90.000,C 0.000} C_DIS
LIN {X 285.372,Y -51.604,Z 115.211,A 169.750,B 90.000,C 0.000} C_DIS
LIN {X 285.317,Y -51.906,Z 115.253,A 169.689,B 90.000,C 0.000} C_DIS
LIN {X 285.306,Y -51.968,Z 115.304,A 169.677,B 90.000,C 0.000} C_DIS
LIN {X 285.298,Y -52.010,Z 115.355,A 169.668,B 90.000,C 0.000} C_DIS
LIN {X 285.261,Y -52.211,Z 115.398,A 169.628,B 90.000,C 0.000} C_DIS
LIN {X 285.246,Y -52.295,Z 115.500,A 169.611,B 90.000,C 0.000} C_DIS
LIN {X 285.209,Y -52.495,Z 115.542,A 169.571,B 90.000,C 0.000} C_DIS
LIN {X 285.201,Y -52.537,Z 115.593,A 169.563,B 90.000,C 0.000} C_DIS
LIN {X 285.190,Y -52.600,Z 115.644,A 169.550,B 90.000,C 0.000} C_DIS
LIN {X 285.134,Y -52.901,Z 115.687,A 169.489,B 90.000,C 0.000} C_DIS
LIN {X 285.123,Y -52.963,Z 115.738,A 169.477,B 90.000,C 0.000} C_DIS
LIN {X 285.115,Y -53.005,Z 115.789,A 169.468,B 90.000,C 0.000} C_DIS
LIN {X 285.077,Y -53.206,Z 115.831,A 169.428,B 90.000,C 0.000} C_DIS
LIN {X 285.070,Y -53.248,Z 115.882,A 169.420,B 90.000,C 0.000} C_DIS
LIN {X 285.058,Y -53.310,Z 115.933,A 169.407,B 90.000,C 0.000} C_DIS
LIN {X 285.001,Y -53.611,Z 115.976,A 169.347,B 90.000,C 0.000} C_DIS
LIN {X 284.990,Y -53.674,Z 116.027,A 169.334,B 90.000,C 0.000} C_DIS
LIN {X 284.982,Y -53.715,Z 116.078,A 169.326,B 90.000,C 0.000} C_DIS
LIN {X 284.944,Y -53.916,Z 116.120,A 169.285,B 90.000,C 0.000} C_DIS
LIN {X 284.928,Y -54.000,Z 116.222,A 169.269,B 90.000,C 0.000} C_DIS
LIN {X 284.890,Y -54.200,Z 116.265,A 169.228,B 90.000,C 0.000} C_DIS
LIN {X 284.882,Y -54.242,Z 116.316,A 169.220,B 90.000,C 0.000} C_DIS
LIN {X 284.870,Y -54.304,Z 116.367,A 169.207,B 90.000,C 0.000} C_DIS
LIN {X 284.813,Y -54.605,Z 116.409,A 169.147,B 90.000,C 0.000} C_DIS
LIN {X 284.801,Y -54.668,Z 116.460,A 169.134,B 90.000,C 0.000} C_DIS
LIN {X 284.793,Y -54.709,Z 116.512,A 169.126,B 90.000,C 0.000} C_DIS
LIN {X 284.754,Y -54.910,Z 116.554,A 169.085,B 90.000,C 0.000} C_DIS
LIN {X 284.738,Y -54.993,Z 116.656,A 169.069,B 90.000,C 0.000} C_DIS
LIN {X 284.699,Y -55.194,Z 116.698,A 169.028,B 90.000,C 0.000} C_DIS
LIN {X 284.691,Y -55.235,Z 116.750,A 169.020,B 90.000,C 0.000} C_DIS
LIN {X 284.679,Y -55.298,Z 116.801,A 169.007,B 90.000,C 0.000} C_DIS
LIN {X 284.620,Y -55.598,Z 116.843,A 168.947,B 90.000,C 0.000} C_DIS
LIN {X 284.608,Y -55.661,Z 116.894,A 168.934,B 90.000,C 0.000} C_DIS
LIN {X 284.600,Y -55.703,Z 116.945,A 168.926,B 90.000,C 0.000} C_DIS
LIN {X 284.561,Y -55.903,Z 116.988,A 168.886,B 90.000,C 0.000} C_DIS
LIN {X 284.544,Y -55.986,Z 117.090,A 168.869,B 90.000,C 0.000} C_DIS
LIN {X 284.505,Y -56.186,Z 117.132,A 168.828,B 90.000,C 0.000} C_DIS
LIN {X 284.497,Y -56.228,Z 117.183,A 168.820,B 90.000,C 0.000} C_DIS
LIN {X 284.484,Y -56.291,Z 117.234,A 168.808,B 90.000,C 0.000} C_DIS
LIN {X 284.425,Y -56.591,Z 117.277,A 168.747,B 90.000,C 0.000} C_DIS
LIN {X 284.412,Y -56.653,Z 117.328,A 168.734,B 90.000,C 0.000} C_DIS
LIN {X 284.404,Y -56.695,Z 117.379,A 168.726,B 90.000,C 0.000} C_DIS
LIN {X 284.364,Y -56.895,Z 117.421,A 168.686,B 90.000,C 0.000} C_DIS
LIN {X 284.347,Y -56.979,Z 117.523,A 168.669,B 90.000,C 0.000} C_DIS
LIN {X 284.307,Y -57.179,Z 117.566,A 168.629,B 90.000,C 0.000} C_DIS
LIN {X 284.299,Y -57.220,Z 117.617,A 168.620,B 90.000,C 0.000} C_DIS
LIN {X 284.286,Y -57.283,Z 117.668,A 168.608,B 90.000,C 0.000} C_DIS
LIN {X 284.226,Y -57.583,Z 117.710,A 168.547,B 90.000,C 0.000} C_DIS
LIN {X 284.213,Y -57.645,Z 117.761,A 168.535,B 90.000,C 0.000} C_DIS
LIN {X 284.205,Y -57.687,Z 117.812,A 168.526,B 90.000,C 0.000} C_DIS
LIN {X 284.164,Y -57.887,Z 117.855,A 168.486,B 90.000,C 0.000} C_DIS
LIN {X 284.155,Y -57.929,Z 117.906,A 168.477,B 90.000,C 0.000} C_DIS
LIN {X 284.143,Y -57.991,Z 117.957,A 168.465,B 90.000,C 0.000} C_DIS
LIN {X 284.081,Y -58.291,Z 117.999,A 168.404,B 90.000,C 0.000} C_DIS
LIN {X 284.068,Y -58.353,Z 118.050,A 168.392,B 90.000,C 0.000} C_DIS
LIN {X 284.060,Y -58.395,Z 118.101,A 168.383,B 90.000,C 0.000} C_DIS
LIN {X 284.019,Y -58.595,Z 118.144,A 168.343,B 90.000,C 0.000} C_DIS
LIN {X 284.002,Y -58.678,Z 118.246,A 168.326,B 90.000,C 0.000} C_DIS
LIN {X 283.960,Y -58.878,Z 118.288,A 168.286,B 90.000,C 0.000} C_DIS
LIN {X 283.952,Y -58.920,Z 118.339,A 168.278,B 90.000,C 0.000} C_DIS
LIN {X 283.939,Y -58.982,Z 118.390,A 168.265,B 90.000,C 0.000} C_DIS
LIN {X 283.876,Y -59.282,Z 118.433,A 168.204,B 90.000,C 0.000} C_DIS
LIN {X 283.863,Y -59.344,Z 118.484,A 168.192,B 90.000,C 0.000} C_DIS
LIN {X 283.854,Y -59.386,Z 118.535,A 168.184,B 90.000,C 0.000} C_DIS
LIN {X 283.813,Y -59.585,Z 118.577,A 168.143,B 90.000,C 0.000} C_DIS
LIN {X 283.795,Y -59.668,Z 118.679,A 168.126,B 90.000,C 0.000} C_DIS
LIN {X 283.753,Y -59.868,Z 118.722,A 168.086,B 90.000,C 0.000} C_DIS
LIN {X 283.744,Y -59.910,Z 118.773,A 168.078,B 90.000,C 0.000} C_DIS
LIN {X 283.731,Y -59.972,Z 118.824,A 168.065,B 90.000,C 0.000} C_DIS
LIN {X 283.668,Y -60.272,Z 118.866,A 168.005,B 90.000,C 0.000} C_DIS
LIN {X 283.654,Y -60.334,Z 118.917,A 167.992,B 90.000,C 0.000} C_DIS
LIN {X 283.646,Y -60.375,Z 118.968,A 167.984,B 90.000,C 0.000} C_DIS
LIN {X 283.603,Y -60.575,Z 119.011,A 167.943,B 90.000,C 0.000} C_DIS
LIN {X 283.585,Y -60.658,Z 119.113,A 167.927,B 90.000,C 0.000} C_DIS
LIN {X 283.542,Y -60.858,Z 119.155,A 167.886,B 90.000,C 0.000} C_DIS
LIN {X 283.534,Y -60.899,Z 119.207,A 167.878,B 90.000,C 0.000} C_DIS
LIN {X 283.520,Y -60.962,Z 119.258,A 167.865,B 90.000,C 0.000} C_DIS
LIN {X 283.456,Y -61.261,Z 119.300,A 167.805,B 90.000,C 0.000} C_DIS
LIN {X 283.442,Y -61.323,Z 119.351,A 167.792,B 90.000,C 0.000} C_DIS
LIN {X 283.433,Y -61.365,Z 119.402,A 167.784,B 90.000,C 0.000} C_DIS
LIN {X 283.390,Y -61.564,Z 119.445,A 167.743,B 90.000,C 0.000} C_DIS
LIN {X 283.381,Y -61.606,Z 119.496,A 167.735,B 90.000,C 0.000} C_DIS
LIN {X 283.367,Y -61.668,Z 119.547,A 167.722,B 90.000,C 0.000} C_DIS
LIN {X 283.302,Y -61.967,Z 119.589,A 167.662,B 90.000,C 0.000} C_DIS
LIN {X 283.289,Y -62.029,Z 119.640,A 167.649,B 90.000,C 0.000} C_DIS
LIN {X 283.279,Y -62.071,Z 119.691,A 167.641,B 90.000,C 0.000} C_DIS
LIN {X 283.236,Y -62.270,Z 119.734,A 167.601,B 90.000,C 0.000} C_DIS
LIN {X 283.217,Y -62.353,Z 119.836,A 167.584,B 90.000,C 0.000} C_DIS
LIN {X 283.173,Y -62.552,Z 119.878,A 167.544,B 90.000,C 0.000} C_DIS
LIN {X 283.164,Y -62.594,Z 119.929,A 167.535,B 90.000,C 0.000} C_DIS
LIN {X 283.151,Y -62.656,Z 119.980,A 167.523,B 90.000,C 0.000} C_DIS
LIN {X 283.084,Y -62.955,Z 120.023,A 167.462,B 90.000,C 0.000} C_DIS
LIN {X 283.070,Y -63.017,Z 120.074,A 167.449,B 90.000,C 0.000} C_DIS
LIN {X 283.061,Y -63.059,Z 120.125,A 167.441,B 90.000,C 0.000} C_DIS
LIN {X 283.017,Y -63.258,Z 120.167,A 167.401,B 90.000,C 0.000} C_DIS
LIN {X 282.998,Y -63.341,Z 120.269,A 167.384,B 90.000,C 0.000} C_DIS
LIN {X 282.954,Y -63.540,Z 120.312,A 167.344,B 90.000,C 0.000} C_DIS
LIN {X 282.944,Y -63.581,Z 120.363,A 167.335,B 90.000,C 0.000} C_DIS
LIN {X 282.930,Y -63.643,Z 120.414,A 167.323,B 90.000,C 0.000} C_DIS
LIN {X 282.863,Y -63.942,Z 120.456,A 167.262,B 90.000,C 0.000} C_DIS
LIN {X 282.849,Y -64.004,Z 120.507,A 167.250,B 90.000,C 0.000} C_DIS
LIN {X 282.839,Y -64.046,Z 120.558,A 167.241,B 90.000,C 0.000} C_DIS
LIN {X 282.794,Y -64.245,Z 120.601,A 167.201,B 90.000,C 0.000} C_DIS
LIN {X 282.775,Y -64.328,Z 120.703,A 167.184,B 90.000,C 0.000} C_DIS
LIN {X 282.730,Y -64.527,Z 120.745,A 167.144,B 90.000,C 0.000} C_DIS
LIN {X 282.721,Y -64.568,Z 120.796,A 167.135,B 90.000,C 0.000} C_DIS
LIN {X 282.706,Y -64.630,Z 120.847,A 167.123,B 90.000,C 0.000} C_DIS
LIN {X 282.638,Y -64.929,Z 120.890,A 167.062,B 90.000,C 0.000} C_DIS
LIN {X 282.624,Y -64.991,Z 120.941,A 167.050,B 90.000,C 0.000} C_DIS
LIN {X 282.614,Y -65.032,Z 120.992,A 167.041,B 90.000,C 0.000} C_DIS
LIN {X 282.568,Y -65.231,Z 121.034,A 167.001,B 90.000,C 0.000} C_DIS
LIN {X 282.549,Y -65.314,Z 121.136,A 166.984,B 90.000,C 0.000} C_DIS
LIN {X 282.503,Y -65.513,Z 121.179,A 166.944,B 90.000,C 0.000} C_DIS
LIN {X 282.494,Y -65.554,Z 121.230,A 166.935,B 90.000,C 0.000} C_DIS
LIN {X 282.479,Y -65.616,Z 121.281,A 166.923,B 90.000,C 0.000} C_DIS
LIN {X 282.410,Y -65.914,Z 121.323,A 166.862,B 90.000,C 0.000} C_DIS
LIN {X 282.395,Y -65.976,Z 121.374,A 166.850,B 90.000,C 0.000} C_DIS
LIN {X 282.386,Y -66.018,Z 121.425,A 166.841,B 90.000,C 0.000} C_DIS
LIN {X 282.339,Y -66.216,Z 121.468,A 166.801,B 90.000,C 0.000} C_DIS
LIN {X 282.320,Y -66.299,Z 121.570,A 166.784,B 90.000,C 0.000} C_DIS
LIN {X 282.273,Y -66.498,Z 121.612,A 166.744,B 90.000,C 0.000} C_DIS
LIN {X 282.263,Y -66.539,Z 121.663,A 166.736,B 90.000,C 0.000} C_DIS
LIN {X 282.249,Y -66.601,Z 121.715,A 166.723,B 90.000,C 0.000} C_DIS
LIN {X 282.178,Y -66.899,Z 121.757,A 166.663,B 90.000,C 0.000} C_DIS
LIN {X 282.163,Y -66.961,Z 121.808,A 166.650,B 90.000,C 0.000} C_DIS
LIN {X 282.154,Y -67.002,Z 121.859,A 166.642,B 90.000,C 0.000} C_DIS
LIN {X 282.106,Y -67.201,Z 121.902,A 166.601,B 90.000,C 0.000} C_DIS
LIN {X 282.097,Y -67.242,Z 121.953,A 166.593,B 90.000,C 0.000} C_DIS
LIN {X 282.082,Y -67.304,Z 122.004,A 166.580,B 90.000,C 0.000} C_DIS
LIN {X 282.011,Y -67.602,Z 122.046,A 166.520,B 90.000,C 0.000} C_DIS
LIN {X 281.996,Y -67.664,Z 122.097,A 166.507,B 90.000,C 0.000} C_DIS
LIN {X 281.986,Y -67.705,Z 122.148,A 166.499,B 90.000,C 0.000} C_DIS
LIN {X 281.938,Y -67.904,Z 122.191,A 166.458,B 90.000,C 0.000} C_DIS
LIN {X 281.918,Y -67.986,Z 122.293,A 166.442,B 90.000,C 0.000} C_DIS
LIN {X 281.870,Y -68.185,Z 122.335,A 166.401,B 90.000,C 0.000} C_DIS
LIN {X 281.860,Y -68.226,Z 122.386,A 166.393,B 90.000,C 0.000} C_DIS
LIN {X 281.845,Y -68.288,Z 122.437,A 166.380,B 90.000,C 0.000} C_DIS
LIN {X 281.773,Y -68.585,Z 122.480,A 166.320,B 90.000,C 0.000} C_DIS
LIN {X 281.758,Y -68.647,Z 122.531,A 166.307,B 90.000,C 0.000} C_DIS
LIN {X 281.748,Y -68.688,Z 122.582,A 166.299,B 90.000,C 0.000} C_DIS
LIN {X 281.700,Y -68.887,Z 122.624,A 166.259,B 90.000,C 0.000} C_DIS
LIN {X 281.679,Y -68.969,Z 122.726,A 166.242,B 90.000,C 0.000} C_DIS
LIN {X 281.631,Y -69.168,Z 122.769,A 166.201,B 90.000,C 0.000} C_DIS
LIN {X 281.621,Y -69.209,Z 122.820,A 166.193,B 90.000,C 0.000} C_DIS
LIN {X 281.605,Y -69.271,Z 122.871,A 166.180,B 90.000,C 0.000} C_DIS
LIN {X 281.532,Y -69.568,Z 122.913,A 166.120,B 90.000,C 0.000} C_DIS
LIN {X 281.517,Y -69.630,Z 122.964,A 166.107,B 90.000,C 0.000} C_DIS
LIN {X 281.507,Y -69.671,Z 123.015,A 166.099,B 90.000,C 0.000} C_DIS
LIN {X 281.457,Y -69.869,Z 123.058,A 166.059,B 90.000,C 0.000} C_DIS
LIN {X 281.447,Y -69.910,Z 123.109,A 166.050,B 90.000,C 0.000} C_DIS
LIN {X 281.432,Y -69.972,Z 123.160,A 166.038,B 90.000,C 0.000} C_DIS
LIN {X 281.358,Y -70.269,Z 123.202,A 165.977,B 90.000,C 0.000} C_DIS
LIN {X 281.342,Y -70.331,Z 123.253,A 165.965,B 90.000,C 0.000} C_DIS
LIN {X 281.332,Y -70.372,Z 123.304,A 165.956,B 90.000,C 0.000} C_DIS
LIN {X 281.282,Y -70.570,Z 123.347,A 165.916,B 90.000,C 0.000} C_DIS
LIN {X 281.262,Y -70.653,Z 123.449,A 165.899,B 90.000,C 0.000} C_DIS
LIN {X 281.212,Y -70.851,Z 123.491,A 165.859,B 90.000,C 0.000} C_DIS
LIN {X 281.202,Y -70.892,Z 123.542,A 165.850,B 90.000,C 0.000} C_DIS
LIN {X 281.186,Y -70.953,Z 123.593,A 165.838,B 90.000,C 0.000} C_DIS
LIN {X 281.111,Y -71.250,Z 123.636,A 165.777,B 90.000,C 0.000} C_DIS
LIN {X 281.095,Y -71.312,Z 123.687,A 165.765,B 90.000,C 0.000} C_DIS
LIN {X 281.085,Y -71.353,Z 123.738,A 165.756,B 90.000,C 0.000} C_DIS
LIN {X 281.035,Y -71.551,Z 123.780,A 165.716,B 90.000,C 0.000} C_DIS
LIN {X 281.014,Y -71.633,Z 123.882,A 165.699,B 90.000,C 0.000} C_DIS
LIN {X 280.963,Y -71.831,Z 123.925,A 165.659,B 90.000,C 0.000} C_DIS
LIN {X 280.953,Y -71.872,Z 123.976,A 165.651,B 90.000,C 0.000} C_DIS
LIN {X 280.937,Y -71.934,Z 124.027,A 165.638,B 90.000,C 0.000} C_DIS
LIN {X 280.861,Y -72.231,Z 124.069,A 165.577,B 90.000,C 0.000} C_DIS
LIN {X 280.845,Y -72.292,Z 124.120,A 165.565,B 90.000,C 0.000} C_DIS
LIN {X 280.834,Y -72.333,Z 124.171,A 165.556,B 90.000,C 0.000} C_DIS
LIN {X 280.783,Y -72.531,Z 124.214,A 165.516,B 90.000,C 0.000} C_DIS
LIN {X 280.762,Y -72.613,Z 124.316,A 165.499,B 90.000,C 0.000} C_DIS
LIN {X 280.711,Y -72.811,Z 124.358,A 165.459,B 90.000,C 0.000} C_DIS
LIN {X 280.700,Y -72.852,Z 124.410,A 165.451,B 90.000,C 0.000} C_DIS
LIN {X 280.684,Y -72.914,Z 124.461,A 165.438,B 90.000,C 0.000} C_DIS
LIN {X 280.607,Y -73.210,Z 124.503,A 165.378,B 90.000,C 0.000} C_DIS
LIN {X 280.591,Y -73.272,Z 124.554,A 165.365,B 90.000,C 0.000} C_DIS
LIN {X 280.580,Y -73.313,Z 124.605,A 165.357,B 90.000,C 0.000} C_DIS
LIN {X 280.529,Y -73.510,Z 124.648,A 165.316,B 90.000,C 0.000} C_DIS
LIN {X 280.507,Y -73.592,Z 124.750,A 165.299,B 90.000,C 0.000} C_DIS
LIN {X 280.455,Y -73.790,Z 124.792,A 165.259,B 90.000,C 0.000} C_DIS
LIN {X 280.444,Y -73.831,Z 124.843,A 165.251,B 90.000,C 0.000} C_DIS
LIN {X 280.428,Y -73.892,Z 124.894,A 165.238,B 90.000,C 0.000} C_DIS
LIN {X 280.350,Y -74.188,Z 124.937,A 165.178,B 90.000,C 0.000} C_DIS
LIN {X 280.334,Y -74.250,Z 124.988,A 165.165,B 90.000,C 0.000} C_DIS
LIN {X 280.323,Y -74.291,Z 125.039,A 165.157,B 90.000,C 0.000} C_DIS
LIN {X 280.270,Y -74.488,Z 125.081,A 165.116,B 90.000,C 0.000} C_DIS
LIN {X 280.259,Y -74.529,Z 125.132,A 165.108,B 90.000,C 0.000} C_DIS
LIN {X 280.243,Y -74.591,Z 125.183,A 165.095,B 90.000,C 0.000} C_DIS
LIN {X 280.164,Y -74.887,Z 125.226,A 165.035,B 90.000,C 0.000} C_DIS
LIN {X 280.148,Y -74.948,Z 125.277,A 165.022,B 90.000,C 0.000} C_DIS
LIN {X 280.137,Y -74.989,Z 125.328,A 165.014,B 90.000,C 0.000} C_DIS
LIN {X 280.084,Y -75.187,Z 125.370,A 164.974,B 90.000,C 0.000} C_DIS
LIN {X 280.062,Y -75.269,Z 125.472,A 164.957,B 90.000,C 0.000} C_DIS
LIN {X 280.009,Y -75.466,Z 125.515,A 164.917,B 90.000,C 0.000} C_DIS
LIN {X 279.998,Y -75.507,Z 125.566,A 164.908,B 90.000,C 0.000} C_DIS
LIN {X 279.981,Y -75.568,Z 125.617,A 164.896,B 90.000,C 0.000} C_DIS
LIN {X 279.901,Y -75.864,Z 125.659,A 164.835,B 90.000,C 0.000} C_DIS
LIN {X 279.885,Y -75.925,Z 125.710,A 164.822,B 90.000,C 0.000} C_DIS
LIN {X 279.873,Y -75.966,Z 125.761,A 164.814,B 90.000,C 0.000} C_DIS
LIN {X 279.820,Y -76.163,Z 125.804,A 164.774,B 90.000,C 0.000} C_DIS
LIN {X 279.798,Y -76.245,Z 125.906,A 164.757,B 90.000,C 0.000} C_DIS
LIN {X 279.744,Y -76.442,Z 125.948,A 164.717,B 90.000,C 0.000} C_DIS
LIN {X 279.733,Y -76.483,Z 125.999,A 164.708,B 90.000,C 0.000} C_DIS
LIN {X 279.716,Y -76.544,Z 126.050,A 164.696,B 90.000,C 0.000} C_DIS
LIN {X 279.635,Y -76.840,Z 126.093,A 164.635,B 90.000,C 0.000} C_DIS
LIN {X 279.618,Y -76.901,Z 126.144,A 164.623,B 90.000,C 0.000} C_DIS
LIN {X 279.607,Y -76.942,Z 126.195,A 164.614,B 90.000,C 0.000} C_DIS
LIN {X 279.552,Y -77.139,Z 126.237,A 164.574,B 90.000,C 0.000} C_DIS
LIN {X 279.530,Y -77.221,Z 126.339,A 164.557,B 90.000,C 0.000} C_DIS
LIN {X 279.475,Y -77.418,Z 126.382,A 164.517,B 90.000,C 0.000} C_DIS
LIN {X 279.464,Y -77.458,Z 126.433,A 164.508,B 90.000,C 0.000} C_DIS
LIN {X 279.447,Y -77.520,Z 126.484,A 164.496,B 90.000,C 0.000} C_DIS
LIN {X 279.365,Y -77.815,Z 126.526,A 164.435,B 90.000,C 0.000} C_DIS
LIN {X 279.348,Y -77.876,Z 126.577,A 164.423,B 90.000,C 0.000} C_DIS
LIN {X 279.337,Y -77.917,Z 126.628,A 164.414,B 90.000,C 0.000} C_DIS
LIN {X 279.282,Y -78.114,Z 126.671,A 164.374,B 90.000,C 0.000} C_DIS
LIN {X 279.259,Y -78.195,Z 126.773,A 164.357,B 90.000,C 0.000} C_DIS
LIN {X 279.204,Y -78.392,Z 126.815,A 164.317,B 90.000,C 0.000} C_DIS
LIN {X 279.192,Y -78.433,Z 126.866,A 164.308,B 90.000,C 0.000} C_DIS
LIN {X 279.175,Y -78.494,Z 126.918,A 164.296,B 90.000,C 0.000} C_DIS
LIN {X 279.092,Y -78.789,Z 126.960,A 164.235,B 90.000,C 0.000} C_DIS
LIN {X 279.075,Y -78.850,Z 127.011,A 164.223,B 90.000,C 0.000} C_DIS
LIN {X 279.063,Y -78.891,Z 127.062,A 164.214,B 90.000,C 0.000} C_DIS
LIN {X 279.007,Y -79.088,Z 127.105,A 164.174,B 90.000,C 0.000} C_DIS
LIN {X 278.996,Y -79.128,Z 127.156,A 164.166,B 90.000,C 0.000} C_DIS
LIN {X 278.979,Y -79.190,Z 127.207,A 164.153,B 90.000,C 0.000} C_DIS
LIN {X 278.895,Y -79.484,Z 127.249,A 164.093,B 90.000,C 0.000} C_DIS
LIN {X 278.877,Y -79.545,Z 127.300,A 164.080,B 90.000,C 0.000} C_DIS
LIN {X 278.866,Y -79.586,Z 127.351,A 164.072,B 90.000,C 0.000} C_DIS
LIN {X 278.810,Y -79.783,Z 127.394,A 164.031,B 90.000,C 0.000} C_DIS
LIN {X 278.786,Y -79.864,Z 127.496,A 164.015,B 90.000,C 0.000} C_DIS
LIN {X 278.730,Y -80.060,Z 127.538,A 163.974,B 90.000,C 0.000} C_DIS
LIN {X 278.718,Y -80.101,Z 127.589,A 163.966,B 90.000,C 0.000} C_DIS
LIN {X 278.701,Y -80.162,Z 127.640,A 163.953,B 90.000,C 0.000} C_DIS
LIN {X 278.616,Y -80.457,Z 127.683,A 163.893,B 90.000,C 0.000} C_DIS
LIN {X 278.598,Y -80.518,Z 127.734,A 163.880,B 90.000,C 0.000} C_DIS
LIN {X 278.586,Y -80.559,Z 127.785,A 163.872,B 90.000,C 0.000} C_DIS
LIN {X 278.529,Y -80.755,Z 127.827,A 163.831,B 90.000,C 0.000} C_DIS
LIN {X 278.506,Y -80.836,Z 127.929,A 163.815,B 90.000,C 0.000} C_DIS
LIN {X 278.449,Y -81.032,Z 127.972,A 163.774,B 90.000,C 0.000} C_DIS
LIN {X 278.437,Y -81.073,Z 128.023,A 163.766,B 90.000,C 0.000} C_DIS
LIN {X 278.419,Y -81.134,Z 128.074,A 163.753,B 90.000,C 0.000} C_DIS
LIN {X 278.333,Y -81.428,Z 128.116,A 163.693,B 90.000,C 0.000} C_DIS
LIN {X 278.315,Y -81.489,Z 128.167,A 163.680,B 90.000,C 0.000} C_DIS
LIN {X 278.304,Y -81.530,Z 128.218,A 163.672,B 90.000,C 0.000} C_DIS
LIN {X 278.246,Y -81.726,Z 128.261,A 163.632,B 90.000,C 0.000} C_DIS
LIN {X 278.222,Y -81.807,Z 128.363,A 163.615,B 90.000,C 0.000} C_DIS
LIN {X 278.164,Y -82.003,Z 128.405,A 163.574,B 90.000,C 0.000} C_DIS
LIN {X 278.152,Y -82.044,Z 128.456,A 163.566,B 90.000,C 0.000} C_DIS
LIN {X 278.134,Y -82.105,Z 128.507,A 163.553,B 90.000,C 0.000} C_DIS
LIN {X 278.048,Y -82.399,Z 128.550,A 163.493,B 90.000,C 0.000} C_DIS
LIN {X 278.030,Y -82.460,Z 128.601,A 163.480,B 90.000,C 0.000} C_DIS
LIN {X 278.017,Y -82.500,Z 128.652,A 163.472,B 90.000,C 0.000} C_DIS
LIN {X 277.959,Y -82.696,Z 128.694,A 163.432,B 90.000,C 0.000} C_DIS
LIN {X 277.947,Y -82.737,Z 128.745,A 163.423,B 90.000,C 0.000} C_DIS
LIN {X 277.929,Y -82.798,Z 128.796,A 163.411,B 90.000,C 0.000} C_DIS
LIN {X 277.841,Y -83.091,Z 128.839,A 163.350,B 90.000,C 0.000} C_DIS
LIN {X 277.823,Y -83.152,Z 128.890,A 163.338,B 90.000,C 0.000} C_DIS
LIN {X 277.811,Y -83.193,Z 128.941,A 163.329,B 90.000,C 0.000} C_DIS
LIN {X 277.752,Y -83.388,Z 128.983,A 163.289,B 90.000,C 0.000} C_DIS
LIN {X 277.728,Y -83.470,Z 129.085,A 163.272,B 90.000,C 0.000} C_DIS
LIN {X 277.669,Y -83.665,Z 129.128,A 163.232,B 90.000,C 0.000} C_DIS
LIN {X 277.657,Y -83.706,Z 129.179,A 163.223,B 90.000,C 0.000} C_DIS
LIN {X 277.638,Y -83.767,Z 129.230,A 163.211,B 90.000,C 0.000} C_DIS
LIN {X 277.550,Y -84.060,Z 129.272,A 163.150,B 90.000,C 0.000} C_DIS
LIN {X 277.531,Y -84.121,Z 129.323,A 163.138,B 90.000,C 0.000} C_DIS
LIN {X 277.519,Y -84.162,Z 129.375,A 163.129,B 90.000,C 0.000} C_DIS
LIN {X 277.460,Y -84.357,Z 129.417,A 163.089,B 90.000,C 0.000} C_DIS
LIN {X 277.435,Y -84.438,Z 129.519,A 163.072,B 90.000,C 0.000} C_DIS
LIN {X 277.376,Y -84.633,Z 129.561,A 163.032,B 90.000,C 0.000} C_DIS
LIN {X 277.363,Y -84.674,Z 129.613,A 163.024,B 90.000,C 0.000} C_DIS
LIN {X 277.345,Y -84.735,Z 129.664,A 163.011,B 90.000,C 0.000} C_DIS
LIN {X 277.255,Y -85.028,Z 129.706,A 162.950,B 90.000,C 0.000} C_DIS
LIN {X 277.236,Y -85.089,Z 129.757,A 162.938,B 90.000,C 0.000} C_DIS
LIN {X 277.224,Y -85.129,Z 129.808,A 162.929,B 90.000,C 0.000} C_DIS
LIN {X 277.164,Y -85.324,Z 129.851,A 162.889,B 90.000,C 0.000} C_DIS
LIN {X 277.139,Y -85.405,Z 129.953,A 162.872,B 90.000,C 0.000} C_DIS
LIN {X 277.079,Y -85.601,Z 129.995,A 162.832,B 90.000,C 0.000} C_DIS
LIN {X 277.066,Y -85.641,Z 130.046,A 162.824,B 90.000,C 0.000} C_DIS
LIN {X 277.047,Y -85.702,Z 130.097,A 162.811,B 90.000,C 0.000} C_DIS
LIN {X 276.957,Y -85.994,Z 130.140,A 162.751,B 90.000,C 0.000} C_DIS
LIN {X 276.938,Y -86.055,Z 130.191,A 162.738,B 90.000,C 0.000} C_DIS
LIN {X 276.925,Y -86.096,Z 130.242,A 162.730,B 90.000,C 0.000} C_DIS
LIN {X 276.864,Y -86.291,Z 130.284,A 162.689,B 90.000,C 0.000} C_DIS
LIN {X 276.839,Y -86.372,Z 130.386,A 162.672,B 90.000,C 0.000} C_DIS
LIN {X 276.778,Y -86.567,Z 130.429,A 162.632,B 90.000,C 0.000} C_DIS
LIN {X 276.766,Y -86.607,Z 130.480,A 162.624,B 90.000,C 0.000} C_DIS
LIN {X 276.747,Y -86.668,Z 130.531,A 162.611,B 90.000,C 0.000} C_DIS
LIN {X 276.655,Y -86.960,Z 130.573,A 162.551,B 90.000,C 0.000} C_DIS
LIN {X 276.636,Y -87.021,Z 130.624,A 162.538,B 90.000,C 0.000} C_DIS
LIN {X 276.623,Y -87.061,Z 130.675,A 162.530,B 90.000,C 0.000} C_DIS
LIN {X 276.562,Y -87.256,Z 130.718,A 162.489,B 90.000,C 0.000} C_DIS
LIN {X 276.549,Y -87.297,Z 130.769,A 162.481,B 90.000,C 0.000} C_DIS
LIN {X 276.530,Y -87.357,Z 130.820,A 162.468,B 90.000,C 0.000} C_DIS
LIN {X 276.437,Y -87.649,Z 130.862,A 162.408,B 90.000,C 0.000} C_DIS
LIN {X 276.418,Y -87.710,Z 130.913,A 162.395,B 90.000,C 0.000} C_DIS
LIN {X 276.405,Y -87.750,Z 130.964,A 162.387,B 90.000,C 0.000} C_DIS
LIN {X 276.343,Y -87.945,Z 131.007,A 162.347,B 90.000,C 0.000} C_DIS
LIN {X 276.318,Y -88.026,Z 131.109,A 162.330,B 90.000,C 0.000} C_DIS
LIN {X 276.256,Y -88.220,Z 131.151,A 162.289,B 90.000,C 0.000} C_DIS
LIN {X 276.243,Y -88.261,Z 131.202,A 162.281,B 90.000,C 0.000} C_DIS
LIN {X 276.223,Y -88.321,Z 131.253,A 162.268,B 90.000,C 0.000} C_DIS
LIN {X 276.130,Y -88.613,Z 131.296,A 162.208,B 90.000,C 0.000} C_DIS
LIN {X 276.110,Y -88.674,Z 131.347,A 162.195,B 90.000,C 0.000} C_DIS
LIN {X 276.097,Y -88.714,Z 131.398,A 162.187,B 90.000,C 0.000} C_DIS
LIN {X 276.035,Y -88.908,Z 131.440,A 162.147,B 90.000,C 0.000} C_DIS
LIN {X 276.009,Y -88.989,Z 131.542,A 162.130,B 90.000,C 0.000} C_DIS
LIN {X 275.946,Y -89.184,Z 131.585,A 162.090,B 90.000,C 0.000} C_DIS
LIN {X 275.933,Y -89.224,Z 131.636,A 162.081,B 90.000,C 0.000} C_DIS
LIN {X 275.914,Y -89.285,Z 131.687,A 162.069,B 90.000,C 0.000} C_DIS
LIN {X 275.819,Y -89.576,Z 131.729,A 162.008,B 90.000,C 0.000} C_DIS
LIN {X 275.799,Y -89.636,Z 131.780,A 161.996,B 90.000,C 0.000} C_DIS
LIN {X 275.786,Y -89.677,Z 131.831,A 161.987,B 90.000,C 0.000} C_DIS
LIN {X 275.723,Y -89.871,Z 131.874,A 161.947,B 90.000,C 0.000} C_DIS
LIN {X 275.697,Y -89.952,Z 131.976,A 161.930,B 90.000,C 0.000} C_DIS
LIN {X 275.633,Y -90.146,Z 132.018,A 161.890,B 90.000,C 0.000} C_DIS
LIN {X 275.620,Y -90.186,Z 132.070,A 161.881,B 90.000,C 0.000} C_DIS
LIN {X 275.600,Y -90.247,Z 132.121,A 161.869,B 90.000,C 0.000} C_DIS
LIN {X 275.505,Y -90.538,Z 132.163,A 161.808,B 90.000,C 0.000} C_DIS
LIN {X 275.485,Y -90.598,Z 132.214,A 161.796,B 90.000,C 0.000} C_DIS
LIN {X 275.472,Y -90.638,Z 132.265,A 161.787,B 90.000,C 0.000} C_DIS
LIN {X 275.408,Y -90.832,Z 132.308,A 161.747,B 90.000,C 0.000} C_DIS
LIN {X 275.381,Y -90.913,Z 132.410,A 161.730,B 90.000,C 0.000} C_DIS
LIN {X 275.317,Y -91.107,Z 132.452,A 161.690,B 90.000,C 0.000} C_DIS
LIN {X 275.304,Y -91.147,Z 132.503,A 161.681,B 90.000,C 0.000} C_DIS
LIN {X 275.284,Y -91.207,Z 132.554,A 161.669,B 90.000,C 0.000} C_DIS
LIN {X 275.187,Y -91.498,Z 132.597,A 161.608,B 90.000,C 0.000} C_DIS
LIN {X 275.167,Y -91.559,Z 132.648,A 161.596,B 90.000,C 0.000} C_DIS
LIN {X 275.154,Y -91.599,Z 132.699,A 161.587,B 90.000,C 0.000} C_DIS
LIN {X 275.089,Y -91.792,Z 132.741,A 161.547,B 90.000,C 0.000} C_DIS
LIN {X 275.076,Y -91.833,Z 132.792,A 161.539,B 90.000,C 0.000} C_DIS
LIN {X 275.056,Y -91.893,Z 132.843,A 161.526,B 90.000,C 0.000} C_DIS
LIN {X 274.959,Y -92.184,Z 132.886,A 161.466,B 90.000,C 0.000} C_DIS
LIN {X 274.938,Y -92.244,Z 132.937,A 161.453,B 90.000,C 0.000} C_DIS
LIN {X 274.925,Y -92.284,Z 132.988,A 161.445,B 90.000,C 0.000} C_DIS
LIN {X 274.860,Y -92.478,Z 133.030,A 161.404,B 90.000,C 0.000} C_DIS
LIN {X 274.833,Y -92.558,Z 133.132,A 161.387,B 90.000,C 0.000} C_DIS
LIN {X 274.767,Y -92.752,Z 133.175,A 161.347,B 90.000,C 0.000} C_DIS
LIN {X 274.754,Y -92.792,Z 133.226,A 161.339,B 90.000,C 0.000} C_DIS
LIN {X 274.733,Y -92.852,Z 133.277,A 161.326,B 90.000,C 0.000} C_DIS
LIN {X 274.635,Y -93.142,Z 133.319,A 161.266,B 90.000,C 0.000} C_DIS
LIN {X 274.615,Y -93.203,Z 133.370,A 161.253,B 90.000,C 0.000} C_DIS
LIN {X 274.601,Y -93.243,Z 133.421,A 161.245,B 90.000,C 0.000} C_DIS
LIN {X 274.535,Y -93.436,Z 133.464,A 161.204,B 90.000,C 0.000} C_DIS
LIN {X 274.508,Y -93.516,Z 133.566,A 161.188,B 90.000,C 0.000} C_DIS
LIN {X 274.442,Y -93.710,Z 133.608,A 161.147,B 90.000,C 0.000} C_DIS
LIN {X 274.428,Y -93.750,Z 133.659,A 161.139,B 90.000,C 0.000} C_DIS
LIN {X 274.408,Y -93.810,Z 133.710,A 161.126,B 90.000,C 0.000} C_DIS
LIN {X 274.309,Y -94.100,Z 133.753,A 161.066,B 90.000,C 0.000} C_DIS
LIN {X 274.288,Y -94.160,Z 133.804,A 161.053,B 90.000,C 0.000} C_DIS
LIN {X 274.274,Y -94.200,Z 133.855,A 161.045,B 90.000,C 0.000} C_DIS
LIN {X 274.208,Y -94.393,Z 133.897,A 161.005,B 90.000,C 0.000} C_DIS
LIN {X 274.180,Y -94.473,Z 133.999,A 160.988,B 90.000,C 0.000} C_DIS
LIN {X 274.114,Y -94.666,Z 134.042,A 160.947,B 90.000,C 0.000} C_DIS
LIN {X 274.100,Y -94.707,Z 134.093,A 160.939,B 90.000,C 0.000} C_DIS
LIN {X 274.079,Y -94.767,Z 134.144,A 160.926,B 90.000,C 0.000} C_DIS
LIN {X 273.979,Y -95.056,Z 134.186,A 160.866,B 90.000,C 0.000} C_DIS
LIN {X 273.958,Y -95.116,Z 134.237,A 160.853,B 90.000,C 0.000} C_DIS
LIN {X 273.944,Y -95.156,Z 134.288,A 160.845,B 90.000,C 0.000} C_DIS
LIN {X 273.877,Y -95.349,Z 134.331,A 160.805,B 90.000,C 0.000} C_DIS
LIN {X 273.863,Y -95.389,Z 134.382,A 160.796,B 90.000,C 0.000} C_DIS
LIN {X 273.842,Y -95.449,Z 134.433,A 160.784,B 90.000,C 0.000} C_DIS
LIN {X 273.741,Y -95.739,Z 134.475,A 160.723,B 90.000,C 0.000} C_DIS
LIN {X 273.720,Y -95.799,Z 134.526,A 160.711,B 90.000,C 0.000} C_DIS
LIN {X 273.706,Y -95.839,Z 134.578,A 160.702,B 90.000,C 0.000} C_DIS
LIN {X 273.638,Y -96.031,Z 134.620,A 160.662,B 90.000,C 0.000} C_DIS
LIN {X 273.610,Y -96.112,Z 134.722,A 160.645,B 90.000,C 0.000} C_DIS
LIN {X 273.543,Y -96.304,Z 134.765,A 160.605,B 90.000,C 0.000} C_DIS
LIN {X 273.528,Y -96.344,Z 134.816,A 160.596,B 90.000,C 0.000} C_DIS
LIN {X 273.507,Y -96.404,Z 134.867,A 160.584,B 90.000,C 0.000} C_DIS
LIN {X 273.405,Y -96.693,Z 134.909,A 160.523,B 90.000,C 0.000} C_DIS
LIN {X 273.384,Y -96.753,Z 134.960,A 160.511,B 90.000,C 0.000} C_DIS
LIN {X 273.370,Y -96.793,Z 135.011,A 160.502,B 90.000,C 0.000} C_DIS
LIN {X 273.302,Y -96.985,Z 135.054,A 160.462,B 90.000,C 0.000} C_DIS
LIN {X 273.273,Y -97.065,Z 135.156,A 160.445,B 90.000,C 0.000} C_DIS
LIN {X 273.205,Y -97.258,Z 135.198,A 160.405,B 90.000,C 0.000} C_DIS
LIN {X 273.191,Y -97.298,Z 135.249,A 160.396,B 90.000,C 0.000} C_DIS
LIN {X 273.169,Y -97.358,Z 135.300,A 160.384,B 90.000,C 0.000} C_DIS
LIN {X 273.066,Y -97.646,Z 135.343,A 160.323,B 90.000,C 0.000} C_DIS
LIN {X 273.045,Y -97.706,Z 135.394,A 160.311,B 90.000,C 0.000} C_DIS
LIN {X 273.031,Y -97.746,Z 135.445,A 160.302,B 90.000,C 0.000} C_DIS
LIN {X 272.962,Y -97.938,Z 135.487,A 160.262,B 90.000,C 0.000} C_DIS
LIN {X 272.933,Y -98.018,Z 135.589,A 160.245,B 90.000,C 0.000} C_DIS
LIN {X 272.864,Y -98.210,Z 135.632,A 160.205,B 90.000,C 0.000} C_DIS
LIN {X 272.850,Y -98.250,Z 135.683,A 160.197,B 90.000,C 0.000} C_DIS
LIN {X 272.828,Y -98.310,Z 135.734,A 160.184,B 90.000,C 0.000} C_DIS
LIN {X 272.724,Y -98.598,Z 135.776,A 160.124,B 90.000,C 0.000} C_DIS
LIN {X 272.702,Y -98.658,Z 135.827,A 160.111,B 90.000,C 0.000} C_DIS
LIN {X 272.688,Y -98.698,Z 135.878,A 160.103,B 90.000,C 0.000} C_DIS
LIN {X 272.618,Y -98.890,Z 135.921,A 160.062,B 90.000,C 0.000} C_DIS
LIN {X 272.604,Y -98.930,Z 135.972,A 160.054,B 90.000,C 0.000} C_DIS
LIN {X 272.582,Y -98.990,Z 136.023,A 160.041,B 90.000,C 0.000} C_DIS
LIN {X 272.477,Y -99.277,Z 136.065,A 159.981,B 90.000,C 0.000} C_DIS
LIN {X 272.456,Y -99.337,Z 136.116,A 159.968,B 90.000,C 0.000} C_DIS
LIN {X 272.441,Y -99.377,Z 136.167,A 159.960,B 90.000,C 0.000} C_DIS
LIN {X 272.371,Y -99.569,Z 136.210,A 159.919,B 90.000,C 0.000} C_DIS
LIN {X 272.342,Y -99.649,Z 136.312,A 159.903,B 90.000,C 0.000} C_DIS
LIN {X 272.272,Y -99.840,Z 136.354,A 159.862,B 90.000,C 0.000} C_DIS
LIN {X 272.257,Y -99.880,Z 136.405,A 159.854,B 90.000,C 0.000} C_DIS
LIN {X 272.235,Y -99.940,Z 136.456,A 159.841,B 90.000,C 0.000} C_DIS
LIN {X 272.129,Y -100.227,Z 136.499,A 159.781,B 90.000,C 0.000} C_DIS
LIN {X 272.107,Y -100.287,Z 136.550,A 159.768,B 90.000,C 0.000} C_DIS
LIN {X 272.093,Y -100.327,Z 136.601,A 159.760,B 90.000,C 0.000} C_DIS
LIN {X 272.022,Y -100.519,Z 136.643,A 159.720,B 90.000,C 0.000} C_DIS
LIN {X 271.993,Y -100.598,Z 136.745,A 159.703,B 90.000,C 0.000} C_DIS
LIN {X 271.922,Y -100.790,Z 136.788,A 159.662,B 90.000,C 0.000} C_DIS
LIN {X 271.907,Y -100.829,Z 136.839,A 159.654,B 90.000,C 0.000} C_DIS
LIN {X 271.885,Y -100.889,Z 136.890,A 159.641,B 90.000,C 0.000} C_DIS
LIN {X 271.778,Y -101.176,Z 136.932,A 159.581,B 90.000,C 0.000} C_DIS
LIN {X 271.756,Y -101.236,Z 136.983,A 159.568,B 90.000,C 0.000} C_DIS
LIN {X 271.741,Y -101.276,Z 137.035,A 159.560,B 90.000,C 0.000} C_DIS
LIN {X 271.670,Y -101.467,Z 137.077,A 159.520,B 90.000,C 0.000} C_DIS
LIN {X 271.640,Y -101.546,Z 137.179,A 159.503,B 90.000,C 0.000} C_DIS
LIN {X 271.569,Y -101.738,Z 137.221,A 159.463,B 90.000,C 0.000} C_DIS
LIN {X 271.554,Y -101.777,Z 137.273,A 159.454,B 90.000,C 0.000} C_DIS
LIN {X 271.531,Y -101.837,Z 137.324,A 159.442,B 90.000,C 0.000} C_DIS
LIN {X 271.424,Y -102.124,Z 137.366,A 159.381,B 90.000,C 0.000} C_DIS
LIN {X 271.401,Y -102.183,Z 137.417,A 159.369,B 90.000,C 0.000} C_DIS
LIN {X 271.386,Y -102.223,Z 137.468,A 159.360,B 90.000,C 0.000} C_DIS
LIN {X 271.314,Y -102.414,Z 137.511,A 159.320,B 90.000,C 0.000} C_DIS
LIN {X 271.284,Y -102.493,Z 137.613,A 159.303,B 90.000,C 0.000} C_DIS
LIN {X 271.212,Y -102.684,Z 137.655,A 159.263,B 90.000,C 0.000} C_DIS
LIN {X 271.197,Y -102.724,Z 137.706,A 159.254,B 90.000,C 0.000} C_DIS
LIN {X 271.174,Y -102.784,Z 137.757,A 159.242,B 90.000,C 0.000} C_DIS
LIN {X 271.066,Y -103.070,Z 137.800,A 159.181,B 90.000,C 0.000} C_DIS
LIN {X 271.043,Y -103.129,Z 137.851,A 159.169,B 90.000,C 0.000} C_DIS
LIN {X 271.028,Y -103.169,Z 137.902,A 159.160,B 90.000,C 0.000} C_DIS
LIN {X 270.955,Y -103.360,Z 137.944,A 159.120,B 90.000,C 0.000} C_DIS
LIN {X 270.940,Y -103.400,Z 137.995,A 159.112,B 90.000,C 0.000} C_DIS
LIN {X 270.917,Y -103.459,Z 138.046,A 159.099,B 90.000,C 0.000} C_DIS
LIN {X 270.808,Y -103.745,Z 138.089,A 159.038,B 90.000,C 0.000} C_DIS
LIN {X 270.785,Y -103.805,Z 138.140,A 159.026,B 90.000,C 0.000} C_DIS
LIN {X 270.770,Y -103.844,Z 138.191,A 159.017,B 90.000,C 0.000} C_DIS
LIN {X 270.697,Y -104.035,Z 138.233,A 158.977,B 90.000,C 0.000} C_DIS
LIN {X 270.666,Y -104.114,Z 138.335,A 158.960,B 90.000,C 0.000} C_DIS
LIN {X 270.593,Y -104.305,Z 138.378,A 158.920,B 90.000,C 0.000} C_DIS
LIN {X 270.578,Y -104.344,Z 138.429,A 158.912,B 90.000,C 0.000} C_DIS
LIN {X 270.555,Y -104.404,Z 138.480,A 158.899,B 90.000,C 0.000} C_DIS
LIN {X 270.444,Y -104.689,Z 138.522,A 158.839,B 90.000,C 0.000} C_DIS
LIN {X 270.421,Y -104.749,Z 138.573,A 158.826,B 90.000,C 0.000} C_DIS
LIN {X 270.406,Y -104.788,Z 138.624,A 158.818,B 90.000,C 0.000} C_DIS
LIN {X 270.332,Y -104.979,Z 138.667,A 158.777,B 90.000,C 0.000} C_DIS
LIN {X 270.301,Y -105.058,Z 138.769,A 158.760,B 90.000,C 0.000} C_DIS
LIN {X 270.227,Y -105.248,Z 138.811,A 158.720,B 90.000,C 0.000} C_DIS
LIN {X 270.212,Y -105.287,Z 138.862,A 158.712,B 90.000,C 0.000} C_DIS
LIN {X 270.189,Y -105.347,Z 138.913,A 158.699,B 90.000,C 0.000} C_DIS
LIN {X 270.133,Y -105.489,Z 138.935,A 158.669,B 90.000,C 0.000} C_DIS
LIN {X 270.054,Y -105.691,Z 138.935,A 158.626,B 90.000,C 0.000} C_DIS
LIN {X 270.062,Y -105.672,Z 139.802,A 158.630,B 90.000,C 0.000} C_DIS
LIN {X 270.081,Y -105.624,Z 139.946,A 158.640,B 90.000,C 0.000} C_DIS
LIN {X 270.099,Y -105.577,Z 140.010,A 158.650,B 90.000,C 0.000} C_DIS
LIN {X 270.118,Y -105.529,Z 140.335,A 158.661,B 90.000,C 0.000} C_DIS
LIN {X 270.160,Y -105.422,Z 140.380,A 158.683,B 90.000,C 0.000} C_DIS
LIN {X 270.197,Y -105.327,Z 140.401,A 158.703,B 90.000,C 0.000} C_DIS
LIN {X 270.227,Y -105.248,Z 140.503,A 158.720,B 90.000,C 0.000} C_DIS
LIN {X 270.301,Y -105.058,Z 140.546,A 158.760,B 90.000,C 0.000} C_DIS
LIN {X 270.317,Y -105.018,Z 140.597,A 158.769,B 90.000,C 0.000} C_DIS
LIN {X 270.340,Y -104.959,Z 140.648,A 158.781,B 90.000,C 0.000} C_DIS
LIN {X 270.451,Y -104.673,Z 140.690,A 158.842,B 90.000,C 0.000} C_DIS
LIN {X 270.474,Y -104.614,Z 140.741,A 158.855,B 90.000,C 0.000} C_DIS
LIN {X 270.489,Y -104.574,Z 140.792,A 158.863,B 90.000,C 0.000} C_DIS
LIN {X 270.562,Y -104.384,Z 140.835,A 158.903,B 90.000,C 0.000} C_DIS
LIN {X 270.593,Y -104.305,Z 140.937,A 158.920,B 90.000,C 0.000} C_DIS
LIN {X 270.666,Y -104.114,Z 140.979,A 158.960,B 90.000,C 0.000} C_DIS
LIN {X 270.682,Y -104.075,Z 141.030,A 158.969,B 90.000,C 0.000} C_DIS
LIN {X 270.704,Y -104.015,Z 141.081,A 158.981,B 90.000,C 0.000} C_DIS
LIN {X 270.814,Y -103.729,Z 141.124,A 159.042,B 90.000,C 0.000} C_DIS
LIN {X 270.837,Y -103.670,Z 141.175,A 159.054,B 90.000,C 0.000} C_DIS
LIN {X 270.852,Y -103.630,Z 141.226,A 159.063,B 90.000,C 0.000} C_DIS
LIN {X 270.925,Y -103.439,Z 141.268,A 159.103,B 90.000,C 0.000} C_DIS
LIN {X 270.955,Y -103.360,Z 141.370,A 159.120,B 90.000,C 0.000} C_DIS
LIN {X 271.028,Y -103.169,Z 141.413,A 159.160,B 90.000,C 0.000} C_DIS
LIN {X 271.043,Y -103.130,Z 141.464,A 159.169,B 90.000,C 0.000} C_DIS
LIN {X 271.066,Y -103.070,Z 141.515,A 159.181,B 90.000,C 0.000} C_DIS
LIN {X 271.174,Y -102.784,Z 141.557,A 159.242,B 90.000,C 0.000} C_DIS
LIN {X 271.197,Y -102.724,Z 141.608,A 159.254,B 90.000,C 0.000} C_DIS
LIN {X 271.212,Y -102.685,Z 141.659,A 159.263,B 90.000,C 0.000} C_DIS
LIN {X 271.284,Y -102.494,Z 141.702,A 159.303,B 90.000,C 0.000} C_DIS
LIN {X 271.314,Y -102.414,Z 141.804,A 159.320,B 90.000,C 0.000} C_DIS
LIN {X 271.386,Y -102.223,Z 141.846,A 159.360,B 90.000,C 0.000} C_DIS
LIN {X 271.401,Y -102.183,Z 141.897,A 159.368,B 90.000,C 0.000} C_DIS
LIN {X 271.424,Y -102.124,Z 141.948,A 159.381,B 90.000,C 0.000} C_DIS
LIN {X 271.531,Y -101.837,Z 141.991,A 159.442,B 90.000,C 0.000} C_DIS
LIN {X 271.554,Y -101.777,Z 142.042,A 159.454,B 90.000,C 0.000} C_DIS
LIN {X 271.568,Y -101.738,Z 142.093,A 159.463,B 90.000,C 0.000} C_DIS
LIN {X 271.640,Y -101.547,Z 142.135,A 159.503,B 90.000,C 0.000} C_DIS
LIN {X 271.670,Y -101.467,Z 142.238,A 159.520,B 90.000,C 0.000} C_DIS
LIN {X 271.741,Y -101.276,Z 142.280,A 159.560,B 90.000,C 0.000} C_DIS
LIN {X 271.756,Y -101.236,Z 142.331,A 159.568,B 90.000,C 0.000} C_DIS
LIN {X 271.778,Y -101.176,Z 142.382,A 159.581,B 90.000,C 0.000} C_DIS
LIN {X 271.885,Y -100.889,Z 142.425,A 159.641,B 90.000,C 0.000} C_DIS
LIN {X 271.907,Y -100.830,Z 142.476,A 159.654,B 90.000,C 0.000} C_DIS
LIN {X 271.922,Y -100.790,Z 142.527,A 159.662,B 90.000,C 0.000} C_DIS
LIN {X 271.993,Y -100.598,Z 142.569,A 159.703,B 90.000,C 0.000} C_DIS
LIN {X 272.022,Y -100.519,Z 142.671,A 159.720,B 90.000,C 0.000} C_DIS
LIN {X 272.093,Y -100.327,Z 142.714,A 159.760,B 90.000,C 0.000} C_DIS
LIN {X 272.107,Y -100.287,Z 142.765,A 159.768,B 90.000,C 0.000} C_DIS
LIN {X 272.129,Y -100.228,Z 142.816,A 159.781,B 90.000,C 0.000} C_DIS
LIN {X 272.235,Y -99.940,Z 142.858,A 159.841,B 90.000,C 0.000} C_DIS
LIN {X 272.257,Y -99.880,Z 142.909,A 159.854,B 90.000,C 0.000} C_DIS
LIN {X 272.272,Y -99.840,Z 142.960,A 159.862,B 90.000,C 0.000} C_DIS
LIN {X 272.342,Y -99.649,Z 143.003,A 159.903,B 90.000,C 0.000} C_DIS
LIN {X 272.371,Y -99.569,Z 143.105,A 159.919,B 90.000,C 0.000} C_DIS
LIN {X 272.441,Y -99.377,Z 143.147,A 159.960,B 90.000,C 0.000} C_DIS
LIN {X 272.456,Y -99.337,Z 143.198,A 159.968,B 90.000,C 0.000} C_DIS
LIN {X 272.477,Y -99.278,Z 143.249,A 159.981,B 90.000,C 0.000} C_DIS
LIN {X 272.582,Y -98.990,Z 143.292,A 160.041,B 90.000,C 0.000} C_DIS
LIN {X 272.604,Y -98.930,Z 143.343,A 160.054,B 90.000,C 0.000} C_DIS
LIN {X 272.618,Y -98.890,Z 143.394,A 160.062,B 90.000,C 0.000} C_DIS
LIN {X 272.688,Y -98.698,Z 143.436,A 160.103,B 90.000,C 0.000} C_DIS
LIN {X 272.717,Y -98.618,Z 143.538,A 160.119,B 90.000,C 0.000} C_DIS
LIN {X 272.786,Y -98.426,Z 143.581,A 160.160,B 90.000,C 0.000} C_DIS
LIN {X 272.801,Y -98.386,Z 143.632,A 160.168,B 90.000,C 0.000} C_DIS
LIN {X 272.822,Y -98.326,Z 143.683,A 160.181,B 90.000,C 0.000} C_DIS
LIN {X 272.926,Y -98.038,Z 143.725,A 160.241,B 90.000,C 0.000} C_DIS
LIN {X 272.947,Y -97.978,Z 143.776,A 160.254,B 90.000,C 0.000} C_DIS
LIN {X 272.962,Y -97.938,Z 143.827,A 160.262,B 90.000,C 0.000} C_DIS
LIN {X 273.031,Y -97.746,Z 143.870,A 160.302,B 90.000,C 0.000} C_DIS
LIN {X 273.059,Y -97.666,Z 143.972,A 160.319,B 90.000,C 0.000} C_DIS
LIN {X 273.128,Y -97.474,Z 144.014,A 160.360,B 90.000,C 0.000} C_DIS
LIN {X 273.142,Y -97.434,Z 144.065,A 160.368,B 90.000,C 0.000} C_DIS
LIN {X 273.164,Y -97.374,Z 144.116,A 160.380,B 90.000,C 0.000} C_DIS
LIN {X 273.266,Y -97.086,Z 144.159,A 160.441,B 90.000,C 0.000} C_DIS
LIN {X 273.287,Y -97.026,Z 144.210,A 160.454,B 90.000,C 0.000} C_DIS
LIN {X 273.302,Y -96.986,Z 144.261,A 160.462,B 90.000,C 0.000} C_DIS
LIN {X 273.370,Y -96.793,Z 144.303,A 160.502,B 90.000,C 0.000} C_DIS
LIN {X 273.398,Y -96.713,Z 144.405,A 160.519,B 90.000,C 0.000} C_DIS
LIN {X 273.466,Y -96.521,Z 144.448,A 160.559,B 90.000,C 0.000} C_DIS
LIN {X 273.480,Y -96.481,Z 144.499,A 160.568,B 90.000,C 0.000} C_DIS
LIN {X 273.502,Y -96.420,Z 144.550,A 160.580,B 90.000,C 0.000} C_DIS
LIN {X 273.603,Y -96.132,Z 144.592,A 160.641,B 90.000,C 0.000} C_DIS
LIN {X 273.624,Y -96.072,Z 144.644,A 160.653,B 90.000,C 0.000} C_DIS
LIN {X 273.638,Y -96.031,Z 144.695,A 160.662,B 90.000,C 0.000} C_DIS
LIN {X 273.706,Y -95.839,Z 144.737,A 160.702,B 90.000,C 0.000} C_DIS
LIN {X 273.734,Y -95.759,Z 144.839,A 160.719,B 90.000,C 0.000} C_DIS
LIN {X 273.801,Y -95.566,Z 144.882,A 160.759,B 90.000,C 0.000} C_DIS
LIN {X 273.815,Y -95.526,Z 144.933,A 160.768,B 90.000,C 0.000} C_DIS
LIN {X 273.836,Y -95.466,Z 144.984,A 160.780,B 90.000,C 0.000} C_DIS
LIN {X 273.937,Y -95.177,Z 145.026,A 160.841,B 90.000,C 0.000} C_DIS
LIN {X 273.958,Y -95.116,Z 145.077,A 160.853,B 90.000,C 0.000} C_DIS
LIN {X 273.972,Y -95.076,Z 145.128,A 160.862,B 90.000,C 0.000} C_DIS
LIN {X 274.039,Y -94.883,Z 145.171,A 160.902,B 90.000,C 0.000} C_DIS
LIN {X 274.066,Y -94.803,Z 145.273,A 160.919,B 90.000,C 0.000} C_DIS
LIN {X 274.133,Y -94.610,Z 145.315,A 160.959,B 90.000,C 0.000} C_DIS
LIN {X 274.161,Y -94.530,Z 145.417,A 160.976,B 90.000,C 0.000} C_DIS
LIN {X 274.227,Y -94.337,Z 145.460,A 161.016,B 90.000,C 0.000} C_DIS
LIN {X 274.241,Y -94.297,Z 145.511,A 161.025,B 90.000,C 0.000} C_DIS
LIN {X 274.262,Y -94.237,Z 145.562,A 161.037,B 90.000,C 0.000} C_DIS
LIN {X 274.361,Y -93.947,Z 145.604,A 161.098,B 90.000,C 0.000} C_DIS
LIN {X 274.382,Y -93.887,Z 145.655,A 161.110,B 90.000,C 0.000} C_DIS
LIN {X 274.395,Y -93.846,Z 145.706,A 161.119,B 90.000,C 0.000} C_DIS
LIN {X 274.461,Y -93.653,Z 145.749,A 161.159,B 90.000,C 0.000} C_DIS
LIN {X 274.475,Y -93.613,Z 145.800,A 161.167,B 90.000,C 0.000} C_DIS
LIN {X 274.496,Y -93.553,Z 145.851,A 161.180,B 90.000,C 0.000} C_DIS
